// TwinCAT 3 PLC project main
// ProgramVersion: 3.1.4024.0
// libraries:
//   Tc2_Standard, * (Beckhoff Automation GmbH)
//   Tc2_System, * (Beckhoff Automation GmbH)
//   Tc3_Module, * (Beckhoff Automation GmbH)
// project tree:
//   / PlcTask.TcTTO
//   POUs/ MAIN.TcPOU, F_ModbusCrc16.TcPOU, FB_EL6022_Port.TcPOU, FB_ModbusRtuMaster.TcPOU, FB_NimServo.TcPOU, FB_PD33.TcPOU, FB_VibrationSensor.TcPOU
//   GVLs/ GVL_PcDemo.TcGVL, GVL_EL6022_IO.TcGVL, GVL_Rs485Demo.TcGVL, GVL_NimServo.TcGVL, GVL_PD33.TcGVL, GVL_Vibration.TcGVL, GVL_ValveIO.TcGVL, GVL_AnalogSensors.TcGVL, GVL_DataLogger.TcGVL
// real-time tasks:
//   TASK PlcTask: cycle T#2ms, priority 20, ADS port 350
// I/O:
//   DEVICE Device 1 (EtherCAT), AmsNetId 172.24.183.94.2.1
//     Term 7 (EK1200) [EK1200-5000 EtherCAT Power supply (2A E-Bus)]
//       Term 2 (EL1008) [EL1008 8Ch. Dig. Input 24V, 3ms]
//       Term 3 (EL2034) [EL2034 4Ch. Dig. Output 24V, 2A, Diagnostic]
//       Term 4 (EL3742) [EL3742 2Ch. Ana. Input 0-20mA, 16bit, DIFF, Oversample]
//       Term 5 (EL3102) [EL3102 2Ch. Ana. Input +/-10V, Diff.]
//       Term 6 (EL6022) [EL6022 Interface 2Ch. (RS422/485)]
//       Term 13 (EL9011) [EL9011 End Terminal]
//   DEVICE Device 4 (USB)
//     Box 1 (CX2100 Power Supply)
//   DEVICE Device 5 (COM Port)
//   DEVICE Device 6 (NOV-DP-RAM)
// variable links:
//   main/main Instance <-> Device 1 (EtherCAT)/Term 7 (EK1200)/Term 4 (EL3742)
//     PlcTask Inputs/GVL_PcDemo.EL3742_Ch2_Sample0_Raw <-> Ch2 Sample 0/Ch2 Value
//     PlcTask Inputs/GVL_AnalogSensors.Pressure_Raw <-> Ch2 Sample 0/Ch2 Value
//     PlcTask Inputs/GVL_AnalogSensors.Torque_Raw <-> Ch1 Sample 0/Ch1 Value
//   main/main Instance <-> Device 1 (EtherCAT)/Term 7 (EK1200)/Term 3 (EL2034)
//     PlcTask Outputs/GVL_ValveIO.Valve{1..4}_Cmd <-> Channel {1..4}/Output  (4 links)
//   main/main Instance <-> Device 1 (EtherCAT)/Term 7 (EK1200)/Term 6 (EL6022)
//     PlcTask Inputs/GVL_EL6022_IO.EL6022_Ch1_DataIn <-> COM Inputs Channel 1/Data In 0
//     PlcTask Inputs/GVL_EL6022_IO.EL6022_Ch2_DataIn <-> COM Inputs Channel 2/Data In 0
//     PlcTask Inputs/GVL_EL6022_IO.EL6022_Ch1_DataIn @bit 8 <-> COM Inputs Channel 1/Data In 1
//     PlcTask Inputs/GVL_EL6022_IO.EL6022_Ch1_DataIn @bit 80 <-> COM Inputs Channel 1/Data In 10
//     PlcTask Inputs/GVL_EL6022_IO.EL6022_Ch1_DataIn @bit 88 <-> COM Inputs Channel 1/Data In 11
//     PlcTask Inputs/GVL_EL6022_IO.EL6022_Ch1_DataIn @bit 96 <-> COM Inputs Channel 1/Data In 12
//     PlcTask Inputs/GVL_EL6022_IO.EL6022_Ch1_DataIn @bit 104 <-> COM Inputs Channel 1/Data In 13
//     PlcTask Inputs/GVL_EL6022_IO.EL6022_Ch1_DataIn @bit 112 <-> COM Inputs Channel 1/Data In 14
//     PlcTask Inputs/GVL_EL6022_IO.EL6022_Ch1_DataIn @bit 120 <-> COM Inputs Channel 1/Data In 15
//     PlcTask Inputs/GVL_EL6022_IO.EL6022_Ch1_DataIn @bit 128 <-> COM Inputs Channel 1/Data In 16
//     PlcTask Inputs/GVL_EL6022_IO.EL6022_Ch1_DataIn @bit 136 <-> COM Inputs Channel 1/Data In 17
//     PlcTask Inputs/GVL_EL6022_IO.EL6022_Ch1_DataIn @bit 144 <-> COM Inputs Channel 1/Data In 18
//     PlcTask Inputs/GVL_EL6022_IO.EL6022_Ch1_DataIn @bit 152 <-> COM Inputs Channel 1/Data In 19
//     PlcTask Inputs/GVL_EL6022_IO.EL6022_Ch1_DataIn @bit 16 <-> COM Inputs Channel 1/Data In 2
//     PlcTask Inputs/GVL_EL6022_IO.EL6022_Ch1_DataIn @bit 160 <-> COM Inputs Channel 1/Data In 20
//     PlcTask Inputs/GVL_EL6022_IO.EL6022_Ch1_DataIn @bit 168 <-> COM Inputs Channel 1/Data In 21
//     PlcTask Inputs/GVL_EL6022_IO.EL6022_Ch1_DataIn @bit 24 <-> COM Inputs Channel 1/Data In 3
//     PlcTask Inputs/GVL_EL6022_IO.EL6022_Ch1_DataIn @bit 32 <-> COM Inputs Channel 1/Data In 4
//     PlcTask Inputs/GVL_EL6022_IO.EL6022_Ch1_DataIn @bit 40 <-> COM Inputs Channel 1/Data In 5
//     PlcTask Inputs/GVL_EL6022_IO.EL6022_Ch1_DataIn @bit 48 <-> COM Inputs Channel 1/Data In 6
//     PlcTask Inputs/GVL_EL6022_IO.EL6022_Ch1_DataIn @bit 56 <-> COM Inputs Channel 1/Data In 7
//     PlcTask Inputs/GVL_EL6022_IO.EL6022_Ch1_DataIn @bit 64 <-> COM Inputs Channel 1/Data In 8
//     PlcTask Inputs/GVL_EL6022_IO.EL6022_Ch1_DataIn @bit 72 <-> COM Inputs Channel 1/Data In 9
//     PlcTask Inputs/GVL_EL6022_IO.EL6022_Ch2_DataIn @bit 8 <-> COM Inputs Channel 2/Data In 1
//     PlcTask Inputs/GVL_EL6022_IO.EL6022_Ch2_DataIn @bit 80 <-> COM Inputs Channel 2/Data In 10
//     PlcTask Inputs/GVL_EL6022_IO.EL6022_Ch2_DataIn @bit 88 <-> COM Inputs Channel 2/Data In 11
//     PlcTask Inputs/GVL_EL6022_IO.EL6022_Ch2_DataIn @bit 96 <-> COM Inputs Channel 2/Data In 12
//     PlcTask Inputs/GVL_EL6022_IO.EL6022_Ch2_DataIn @bit 104 <-> COM Inputs Channel 2/Data In 13
//     PlcTask Inputs/GVL_EL6022_IO.EL6022_Ch2_DataIn @bit 112 <-> COM Inputs Channel 2/Data In 14
//     PlcTask Inputs/GVL_EL6022_IO.EL6022_Ch2_DataIn @bit 120 <-> COM Inputs Channel 2/Data In 15
//     PlcTask Inputs/GVL_EL6022_IO.EL6022_Ch2_DataIn @bit 128 <-> COM Inputs Channel 2/Data In 16
//     PlcTask Inputs/GVL_EL6022_IO.EL6022_Ch2_DataIn @bit 136 <-> COM Inputs Channel 2/Data In 17
//     PlcTask Inputs/GVL_EL6022_IO.EL6022_Ch2_DataIn @bit 144 <-> COM Inputs Channel 2/Data In 18
//     PlcTask Inputs/GVL_EL6022_IO.EL6022_Ch2_DataIn @bit 152 <-> COM Inputs Channel 2/Data In 19
//     PlcTask Inputs/GVL_EL6022_IO.EL6022_Ch2_DataIn @bit 16 <-> COM Inputs Channel 2/Data In 2
//     PlcTask Inputs/GVL_EL6022_IO.EL6022_Ch2_DataIn @bit 160 <-> COM Inputs Channel 2/Data In 20
//     PlcTask Inputs/GVL_EL6022_IO.EL6022_Ch2_DataIn @bit 168 <-> COM Inputs Channel 2/Data In 21
//     PlcTask Inputs/GVL_EL6022_IO.EL6022_Ch2_DataIn @bit 24 <-> COM Inputs Channel 2/Data In 3
//     PlcTask Inputs/GVL_EL6022_IO.EL6022_Ch2_DataIn @bit 32 <-> COM Inputs Channel 2/Data In 4
//     PlcTask Inputs/GVL_EL6022_IO.EL6022_Ch2_DataIn @bit 40 <-> COM Inputs Channel 2/Data In 5
//     PlcTask Inputs/GVL_EL6022_IO.EL6022_Ch2_DataIn @bit 48 <-> COM Inputs Channel 2/Data In 6
//     PlcTask Inputs/GVL_EL6022_IO.EL6022_Ch2_DataIn @bit 56 <-> COM Inputs Channel 2/Data In 7
//     PlcTask Inputs/GVL_EL6022_IO.EL6022_Ch2_DataIn @bit 64 <-> COM Inputs Channel 2/Data In 8
//     PlcTask Inputs/GVL_EL6022_IO.EL6022_Ch2_DataIn @bit 72 <-> COM Inputs Channel 2/Data In 9
//     PlcTask Inputs/GVL_EL6022_IO.EL6022_Ch1_Status <-> COM Inputs Channel 1/Status
//     PlcTask Inputs/GVL_EL6022_IO.EL6022_Ch2_Status <-> COM Inputs Channel 2/Status
//     PlcTask Outputs/GVL_EL6022_IO.EL6022_Ch1_Ctrl <-> COM Outputs Channel 1/Ctrl
//     PlcTask Outputs/GVL_EL6022_IO.EL6022_Ch2_Ctrl <-> COM Outputs Channel 2/Ctrl
//     PlcTask Outputs/GVL_EL6022_IO.EL6022_Ch1_DataOut <-> COM Outputs Channel 1/Data Out 0
//     PlcTask Outputs/GVL_EL6022_IO.EL6022_Ch2_DataOut <-> COM Outputs Channel 2/Data Out 0
//     PlcTask Outputs/GVL_EL6022_IO.EL6022_Ch1_DataOut @bit 8 <-> COM Outputs Channel 1/Data Out 1
//     PlcTask Outputs/GVL_EL6022_IO.EL6022_Ch1_DataOut @bit 80 <-> COM Outputs Channel 1/Data Out 10
//     PlcTask Outputs/GVL_EL6022_IO.EL6022_Ch1_DataOut @bit 88 <-> COM Outputs Channel 1/Data Out 11
//     PlcTask Outputs/GVL_EL6022_IO.EL6022_Ch1_DataOut @bit 96 <-> COM Outputs Channel 1/Data Out 12
//     PlcTask Outputs/GVL_EL6022_IO.EL6022_Ch1_DataOut @bit 104 <-> COM Outputs Channel 1/Data Out 13
//     PlcTask Outputs/GVL_EL6022_IO.EL6022_Ch1_DataOut @bit 112 <-> COM Outputs Channel 1/Data Out 14
//     PlcTask Outputs/GVL_EL6022_IO.EL6022_Ch1_DataOut @bit 120 <-> COM Outputs Channel 1/Data Out 15
//     PlcTask Outputs/GVL_EL6022_IO.EL6022_Ch1_DataOut @bit 128 <-> COM Outputs Channel 1/Data Out 16
//     PlcTask Outputs/GVL_EL6022_IO.EL6022_Ch1_DataOut @bit 136 <-> COM Outputs Channel 1/Data Out 17
//     PlcTask Outputs/GVL_EL6022_IO.EL6022_Ch1_DataOut @bit 144 <-> COM Outputs Channel 1/Data Out 18
//     PlcTask Outputs/GVL_EL6022_IO.EL6022_Ch1_DataOut @bit 152 <-> COM Outputs Channel 1/Data Out 19
//     PlcTask Outputs/GVL_EL6022_IO.EL6022_Ch1_DataOut @bit 16 <-> COM Outputs Channel 1/Data Out 2
//     PlcTask Outputs/GVL_EL6022_IO.EL6022_Ch1_DataOut @bit 160 <-> COM Outputs Channel 1/Data Out 20
//     PlcTask Outputs/GVL_EL6022_IO.EL6022_Ch1_DataOut @bit 168 <-> COM Outputs Channel 1/Data Out 21
//     PlcTask Outputs/GVL_EL6022_IO.EL6022_Ch1_DataOut @bit 24 <-> COM Outputs Channel 1/Data Out 3
//     PlcTask Outputs/GVL_EL6022_IO.EL6022_Ch1_DataOut @bit 32 <-> COM Outputs Channel 1/Data Out 4
//     PlcTask Outputs/GVL_EL6022_IO.EL6022_Ch1_DataOut @bit 40 <-> COM Outputs Channel 1/Data Out 5
//     PlcTask Outputs/GVL_EL6022_IO.EL6022_Ch1_DataOut @bit 48 <-> COM Outputs Channel 1/Data Out 6
//     PlcTask Outputs/GVL_EL6022_IO.EL6022_Ch1_DataOut @bit 56 <-> COM Outputs Channel 1/Data Out 7
//     PlcTask Outputs/GVL_EL6022_IO.EL6022_Ch1_DataOut @bit 64 <-> COM Outputs Channel 1/Data Out 8
//     PlcTask Outputs/GVL_EL6022_IO.EL6022_Ch1_DataOut @bit 72 <-> COM Outputs Channel 1/Data Out 9
//     PlcTask Outputs/GVL_EL6022_IO.EL6022_Ch2_DataOut @bit 8 <-> COM Outputs Channel 2/Data Out 1
//     PlcTask Outputs/GVL_EL6022_IO.EL6022_Ch2_DataOut @bit 80 <-> COM Outputs Channel 2/Data Out 10
//     PlcTask Outputs/GVL_EL6022_IO.EL6022_Ch2_DataOut @bit 88 <-> COM Outputs Channel 2/Data Out 11
//     PlcTask Outputs/GVL_EL6022_IO.EL6022_Ch2_DataOut @bit 96 <-> COM Outputs Channel 2/Data Out 12
//     PlcTask Outputs/GVL_EL6022_IO.EL6022_Ch2_DataOut @bit 104 <-> COM Outputs Channel 2/Data Out 13
//     PlcTask Outputs/GVL_EL6022_IO.EL6022_Ch2_DataOut @bit 112 <-> COM Outputs Channel 2/Data Out 14
//     PlcTask Outputs/GVL_EL6022_IO.EL6022_Ch2_DataOut @bit 120 <-> COM Outputs Channel 2/Data Out 15
//     PlcTask Outputs/GVL_EL6022_IO.EL6022_Ch2_DataOut @bit 128 <-> COM Outputs Channel 2/Data Out 16
//     PlcTask Outputs/GVL_EL6022_IO.EL6022_Ch2_DataOut @bit 136 <-> COM Outputs Channel 2/Data Out 17
//     PlcTask Outputs/GVL_EL6022_IO.EL6022_Ch2_DataOut @bit 144 <-> COM Outputs Channel 2/Data Out 18
//     PlcTask Outputs/GVL_EL6022_IO.EL6022_Ch2_DataOut @bit 152 <-> COM Outputs Channel 2/Data Out 19
//     PlcTask Outputs/GVL_EL6022_IO.EL6022_Ch2_DataOut @bit 16 <-> COM Outputs Channel 2/Data Out 2
//     PlcTask Outputs/GVL_EL6022_IO.EL6022_Ch2_DataOut @bit 160 <-> COM Outputs Channel 2/Data Out 20
//     PlcTask Outputs/GVL_EL6022_IO.EL6022_Ch2_DataOut @bit 168 <-> COM Outputs Channel 2/Data Out 21
//     PlcTask Outputs/GVL_EL6022_IO.EL6022_Ch2_DataOut @bit 24 <-> COM Outputs Channel 2/Data Out 3
//     PlcTask Outputs/GVL_EL6022_IO.EL6022_Ch2_DataOut @bit 32 <-> COM Outputs Channel 2/Data Out 4
//     PlcTask Outputs/GVL_EL6022_IO.EL6022_Ch2_DataOut @bit 40 <-> COM Outputs Channel 2/Data Out 5
//     PlcTask Outputs/GVL_EL6022_IO.EL6022_Ch2_DataOut @bit 48 <-> COM Outputs Channel 2/Data Out 6
//     PlcTask Outputs/GVL_EL6022_IO.EL6022_Ch2_DataOut @bit 56 <-> COM Outputs Channel 2/Data Out 7
//     PlcTask Outputs/GVL_EL6022_IO.EL6022_Ch2_DataOut @bit 64 <-> COM Outputs Channel 2/Data Out 8
//     PlcTask Outputs/GVL_EL6022_IO.EL6022_Ch2_DataOut @bit 72 <-> COM Outputs Channel 2/Data Out 9

CONFIGURATION main
    RESOURCE PLC ON TwinCAT3
        TASK PlcTask(INTERVAL := T#2ms, PRIORITY := 20);
        PROGRAM MAIN WITH PlcTask : MAIN;
    END_RESOURCE
END_CONFIGURATION

// ---- GVLs/GVL_PcDemo.TcGVL
VAR_GLOBAL
    (*
      Demo input to be linked in TwinCAT I/O mapping:
      EL3742 -> Ch2 Sample 0 -> Ch2 Value
    *)
    EL3742_Ch2_Sample0_Raw AT %I*: INT;

    (*
      PLC-side copy / heartbeat for ADS reads.
    *)
    EL3742_Ch2_Sample0_RawCopy : INT;
    MainCycleCounter : ULINT;
END_VAR

// ---- GVLs/GVL_EL6022_IO.TcGVL
VAR_GLOBAL
    (*
      EL6022 process data mapping placeholders.
      Map these in TwinCAT I/O Mapping to:
        Term 6 (EL6022) -> COM Inputs/Outputs Channel 1/2
      Notes:
        - Status/Ctrl are WORD. Typically: low byte = flags, high byte = length (bytes).
        - Data arrays are 22 bytes (0..21).
    *)

    // Channel 1
    EL6022_Ch1_Status AT %I* : WORD;
    EL6022_Ch1_DataIn AT %I* : ARRAY [0..21] OF USINT;

    EL6022_Ch1_Ctrl AT %Q* : WORD;
    EL6022_Ch1_DataOut AT %Q* : ARRAY [0..21] OF USINT;

    // Channel 2
    EL6022_Ch2_Status AT %I* : WORD;
    EL6022_Ch2_DataIn AT %I* : ARRAY [0..21] OF USINT;

    EL6022_Ch2_Ctrl AT %Q* : WORD;
    EL6022_Ch2_DataOut AT %Q* : ARRAY [0..21] OF USINT;
END_VAR

// ---- GVLs/GVL_Rs485Demo.TcGVL
VAR_GLOBAL
    (*
      PC <-> PLC demo interface for EL6022 RS-485 loopback testing.
      PC writes Tx* and increments TxSeq.
      PLC sends via selected channel and exposes last Rx* from either channel.
    *)

    Enable : BOOL; // Enable demo logic in MAIN (avoid conflicts with real device drivers)

    TxSeq : UDINT;
    TxUseCh2 : BOOL; // FALSE => TX on Ch1, TRUE => TX on Ch2
    TxLen : USINT;
    TxData : ARRAY [0..21] OF USINT;

    TxBusy : BOOL;
    TxDoneSeq : UDINT;
    TxError : UDINT;

    RxSeq : UDINT;
    RxFromCh2 : BOOL;
    RxLen : USINT;
    RxStatus : WORD;
    RxData : ARRAY [0..21] OF USINT;

    Debug_Ch1_Status : WORD;
    Debug_Ch2_Status : WORD;
    Debug_Ch1_Ctrl : WORD;
    Debug_Ch2_Ctrl : WORD;
END_VAR

// ---- GVLs/GVL_NimServo.TcGVL
VAR_GLOBAL
    (*
      NiMotion servo host interface (Modbus RTU over EL6022 / RS-485).

      Notes:
      - PLC implements Modbus + servo control. PC only uses ADS to write macro-level commands and read telemetry.
      - Channel selects EL6022 channel 1/2.
      - WordSwap32 can be used to adapt 32-bit register word order if needed.
    *)

    Enable : BOOL;
    Channel : USINT := 1; // 1 or 2
    SlaveId : USINT := 1; // Modbus address 1..247

    AutoSetCia402Mode : BOOL := TRUE; // Write I2002-1 (H00B1) to 0 if needed

    DesiredMode : USINT := 2; // 2=VM, 9=CSV
    PowerEnable : BOOL;
    TargetVelocity : DINT; // Raw target velocity (unit depends on drive configuration)
    WordSwap32 : BOOL;
    TestForceVelocityWrite : BOOL; // Debug: send 60FF write even without successful comms / OP enabled
    ExtendedPoll : BOOL := TRUE;    // TRUE: poll extended diagnostics (more traffic, more risk of timeouts on noisy links)
    ApplyVmConfig : BOOL := FALSE;  // TRUE: apply VM min/max/accel/decel params via Modbus when PowerEnable=FALSE

    // VM mode parameters (from Modbus.db)
    VmSpeedMinRpm : UDINT := 0;     // I6046-1 (H0385), 32-bit
    VmSpeedMaxRpm : UDINT := 500;   // I6046-2 (H0387), 32-bit
    VmAccelRpm : UDINT := 200;      // I6048-1 (H0389), 32-bit
    VmAccelTimeS : UINT := 1;       // I6048-2 (H038B), 16-bit, seconds
    VmDecelRpm : UDINT := 200;      // I6049-1 (H038C), 32-bit
    VmDecelTimeS : UINT := 1;       // I6049-2 (H038E), 16-bit, seconds

    CmdSeq : UDINT; // PC increments to request a one-shot command
    Cmd : USINT;    // 0=None, 1=FaultReset

    CmdAckSeq : UDINT;
    Busy : BOOL;
    CommOk : BOOL;
    CommErrorCount : UDINT;
    LastErrorId : UDINT;

    // Telemetry (raw registers)
    ControlMode : USINT;      // I2002-1 (H00B1): 0=CIA402
    ControlModeOk : BOOL;
    StatusWord : UINT;         // 6041 (H0381)
    ControlWord : UINT;        // last written 6040 (H0380)

    // Diagnostics / preconditions
    Cia402State : USINT;       // 0=Unknown, 1=NotReady, 2=SwitchOnDisabled, 3=Ready, 4=SwitchedOn, 5=OpEnabled, 6=FaultReaction, 7=Fault, 8=QuickStop
    ErrorRegister : USINT;     // I1001 (H0000) low byte
    CurrentAlarm : USINT;      // I1003-0 (H0001) low byte

    DiSignals : UINT;          // I200B-5 (H01E2), raw DI monitor bits
    DoSignals : UINT;          // I200B-6 (H01E3), raw DO monitor bits
    DcBusVoltage : UINT;       // I200B-21 (H01F7), bus voltage (unit per drive)
    ModuleTemp : INT;          // I200B-22 (H01F8), module temperature (unit per drive)

    Di1Func : USINT;           // I2003-3 (H00D5) low byte
    Di1Logic : USINT;          // I2003-4 (H00D6) low byte
    Di2Func : USINT;           // I2003-5 (H00D7) low byte
    Di2Logic : USINT;          // I2003-6 (H00D8) low byte
    Di3Func : USINT;           // I2003-7 (H00D9) low byte
    Di3Logic : USINT;          // I2003-8 (H00DA) low byte
    Di4Func : USINT;           // I2003-9 (H00DB) low byte
    Di4Logic : USINT;          // I2003-10 (H00DC) low byte
    Di5Func : USINT;           // I2003-11 (H00DD) low byte
    Di5Logic : USINT;          // I2003-12 (H00DE) low byte
    Di6Func : USINT;           // I2003-13 (H00DF) low byte
    Di6Logic : USINT;          // I2003-14 (H00E0) low byte
    Di7Func : USINT;           // I2003-15 (H00E1) low byte
    Di7Logic : USINT;          // I2003-16 (H00E2) low byte
    Di8Func : USINT;           // I2003-17 (H00E3) low byte
    Di8Logic : USINT;          // I2003-18 (H00E4) low byte
    Di9Func : USINT;           // I2003-19 (H00E5) low byte
    Di9Logic : USINT;          // I2003-20 (H00E6) low byte

    EnableDiIndex : USINT;     // 0=None, 1..9 = which DI is "Enable(1)"
    EnableDiRequired : BOOL;   // EnableDiIndex <> 0
    EnableDiActive : BOOL;     // Computed from DiSignals + selected DI logic when required
    EnableDiOk : BOOL;         // NOT EnableDiRequired OR EnableDiActive

    // Drive status (vendor-specific)
    DriveInternalState : USINT; // I200B-1 (H01DE), see Modbus.db selects (0=未准备好, 1=准备好, 8=速度闭环控制...)
    FpgaSystemStatus : UINT;    // I200B-24 (H01FA)
    FpgaSystemFault : UINT;     // I200B-25 (H01FB)
    EncoderInternalFault : UINT; // I200B-26 (H01FC) 编码内部故障信息
    FaultRecord : UINT;         // I200B-27 (H01FD)
    AbsEncoderWord : UINT;      // I200B-23 (H01F9) FPGA给出绝对编码

    ModeDisplay : USINT;       // 6061 (H03C3) low byte
    ActualVelocity : DINT;     // 606C (H03D5)
    ActualPosition : DINT;     // 6064 (H03C8)
    CurrentFeedback : INT;     // 6078 (H03E4)

    // VM mode telemetry (from Modbus.db)
    VmTargetSpeedRpm : INT;    // I6042 (H0382) 16-bit
    VmTargetSpeedEffRpm : INT; // I6043 (H0383) 16-bit (effective)
    VmActualSpeedRpm : INT;    // I6044 (H0384) 16-bit

    // VM config progress (helps debug/avoid powering on before config is applied)
    VmCfgPending : BOOL;
    VmCfgIndex : USINT;

    // Debug frames
    LastTxLen : USINT;
    LastTx : ARRAY [0..21] OF USINT;
    LastRxLen : USINT;
    LastRx : ARRAY [0..21] OF USINT;
END_VAR

// ---- GVLs/GVL_PD33.TcGVL
VAR_GLOBAL
    (*
      PD33 series laser displacement sensor (Modbus RTU over EL6022 / RS-485).

      Registers (from manual screenshots):
      Current mode: passive parsing of PD33 full-speed active output.
      Expected frame: slave=1, function=3, bytecount=4, payload i32 low-word-first, CRC16.
      Scale: raw / 1000.0 = mm.
    *)

    Enable : BOOL;
    Channel : USINT := 1; // 1 or 2 (EL6022 channel)
    SlaveId : USINT := 1; // Modbus address

    // PD33 frames shown in the manual interpret 32-bit values as "low word first".
    // Keep this TRUE unless you verify your device uses the opposite order.
    WordSwap32 : BOOL := TRUE;
    UseDisplayRegister3B : BOOL := FALSE; // reserved; passive full-speed output parser does not send read requests

    // Command handshake (PC writes Cmd+CmdSeq; PLC sets CmdAckSeq after completion)
    CmdSeq : UDINT;
    Cmd : USINT; // reserved in passive mode
    CmdAckSeq : UDINT;
    Busy : BOOL;

    // Diagnostics
    ChannelConflict : BOOL; // TRUE when another driver is using the same EL6022 channel
    PortReady : BOOL;
    CommOk : BOOL;
    CommErrorCount : UDINT;
    LastErrorId : UDINT;
    ExceptionCode : USINT;
    RxDiscardCount : UDINT;
    LastDiscardId : UDINT;

    // Measurements
    AbsRaw : DINT; // raw units depend on UseDisplayRegister3B
    RelRaw : DINT; // raw units depend on UseDisplayRegister3B
    AbsMm : LREAL; // computed
    RelMm : LREAL; // computed

    ZeroWord : UINT; // last written value to 0x0020 (for debug)

    // Debug frames (last Modbus tx/rx)
    LastTxLen : USINT;
    LastTx : ARRAY [0..21] OF USINT;
    LastRxLen : USINT;
    LastRx : ARRAY [0..21] OF USINT;
END_VAR

// ---- GVLs/GVL_Vibration.TcGVL
VAR_GLOBAL
    (*
      VB02/WTVB02-485 vibration sensor over EL6022 Channel 2.

      SDK register map:
        0x34..0x36 vibration acceleration X/Y/Z, raw INT, scale raw / 32768 * 16
        0x3A..0x3C vibration velocity X/Y/Z, raw INT, scale raw / 100
        0x40      temperature, raw INT, scale raw / 100
        0x41..0x43 displacement X/Y/Z, raw INT
        0x44..0x46 frequency X/Y/Z, raw INT, scale raw / 10

      EL6022 frame limit is 22 bytes, so PLC reads these as 3 Modbus transactions.
    *)

    Enable : BOOL := FALSE;
    Channel : USINT := 2;
    SlaveId : USINT := 16#50;
    MinGapMs : UINT := 200;
    TimeoutMs : UINT := 500;

    Busy : BOOL;
    PortReady : BOOL;
    CommOk : BOOL;
    CommErrorCount : UDINT;
    LastErrorId : UDINT;
    ExceptionCode : USINT;
    RxDiscardCount : UDINT;
    LastDiscardId : UDINT;
    SampleSeq : UDINT;

    AccXRaw : INT;
    AccYRaw : INT;
    AccZRaw : INT;
    VelXRaw : INT;
    VelYRaw : INT;
    VelZRaw : INT;
    TempRaw : INT;
    DispXRaw : INT;
    DispYRaw : INT;
    DispZRaw : INT;
    FreqXRaw : INT;
    FreqYRaw : INT;
    FreqZRaw : INT;

    AccX : LREAL;
    AccY : LREAL;
    AccZ : LREAL;
    VelX : LREAL;
    VelY : LREAL;
    VelZ : LREAL;
    TempC : LREAL;
    DispX : LREAL;
    DispY : LREAL;
    DispZ : LREAL;
    FreqX : LREAL;
    FreqY : LREAL;
    FreqZ : LREAL;

    LastTxLen : USINT;
    LastTx : ARRAY [0..21] OF USINT;
    LastRxLen : USINT;
    LastRx : ARRAY [0..21] OF USINT;
END_VAR

// ---- GVLs/GVL_ValveIO.TcGVL
VAR_GLOBAL
    (*
      Valve digital outputs placeholder.

      Hardware: Term 3 (EL2034) 4Ch. Digital Output.

      Map in TwinCAT I/O mapping:
        EL2034 -> Channel 1 -> Output  => Valve1_Cmd
        EL2034 -> Channel 2 -> Output  => Valve2_Cmd
        EL2034 -> Channel 3 -> Output  => Valve3_Cmd
        EL2034 -> Channel 4 -> Output  => Valve4_Cmd

      Notes:
        - Use AT %Q* so the symbol shows up in "Link To..." list.
        - Valve*_Fb are software feedback mirrors (what PLC currently drives).
    *)

    Valve1_Cmd AT %Q* : BOOL;
    Valve2_Cmd AT %Q* : BOOL;
    Valve3_Cmd AT %Q* : BOOL;
    Valve4_Cmd AT %Q* : BOOL;

    Valve1_Fb : BOOL;
    Valve2_Fb : BOOL;
    Valve3_Fb : BOOL;
    Valve4_Fb : BOOL;

    // Master enable for all valve outputs (safety interlock).
    Enable : BOOL := FALSE;
END_VAR

// ---- GVLs/GVL_AnalogSensors.TcGVL
VAR_GLOBAL
    (*
      Analog current sampling (EL3742 2Ch 0-20mA) placeholders.

      Map in TwinCAT I/O mapping:
        EL3742 -> Ch2 Sample 0 -> Ch2 Value => Pressure_Raw
        EL3742 -> Ch1 Sample 0 -> Ch1 Value => Torque_Raw

      Raw type follows EL3742 PDO type (INT16).
    *)

    Pressure_Raw AT %I* : INT;
    Torque_Raw AT %I* : INT;

    // PLC-side copies for ADS reads / snapshot.
    Pressure_RawCopy : INT;
    Torque_RawCopy : INT;
END_VAR

// ---- GVLs/GVL_DataLogger.TcGVL
VAR_GLOBAL
    (*
      PLC-side ring buffer logger to avoid ADS per-sample reads.

      Design:
        - MAIN (2ms task) writes a fixed-size record into a byte ring buffer.
        - PC reads Head and Buffer bytes via ADS and reconstructs records.
        - If PC is too slow and overrun happens, OverrunCount increments.

      Record layout (little-endian):
        u32 magic = 0x56424D31 ('VBM1')
        u32 seq
        u32 t_us (monotonic from cycle count * 2000us)
        i16 pressure_raw
        i16 torque_raw
        i32 pd33_abs_raw
        i32 pd33_rel_raw
        i16 vib_acc_x_raw
        i16 vib_acc_y_raw
        i16 vib_acc_z_raw
        i16 vib_vel_x_raw
        i16 vib_vel_y_raw
        i16 vib_vel_z_raw
        i16 vib_temp_raw
        i16 vib_disp_x_raw
        i16 vib_disp_y_raw
        i16 vib_disp_z_raw
        i16 vib_freq_x_raw
        i16 vib_freq_y_raw
        i16 vib_freq_z_raw
        u8  valves (bit0..3)
        u8  flags (bit0=pd33_comm_ok, bit1=vibration_comm_ok)
        u16 reserved
      Total: 54 bytes per record
    *)

    Enable : BOOL := FALSE;
    Reset : BOOL := FALSE;

    // Ring buffer state (byte indices)
    Head : UDINT; // next write index (monotonic, wraps by modulo on read side)
    Tail : UDINT; // PC should update this as "consumed" index to prevent Overrun

    OverrunCount : UDINT;
    DropCount : UDINT;

    Seq : UDINT;

    // Constants
    RecordSize : UDINT := 54;
    BufferSize : UDINT := 54 * 4096; // 221,184 bytes (~8.2s at 500Hz)

    Buffer : ARRAY [0..(54*4096)-1] OF USINT;
END_VAR

// ---- POUs/MAIN.TcPOU
PROGRAM MAIN
VAR
    initCh1Done : BOOL;
    initCh2Done : BOOL;
    fbNimServo : FB_NimServo;
    fbPd33 : FB_PD33;
    fbVibration : FB_VibrationSensor;

    // DataLogger internal (packed ring buffer)
    logResetLatched : BOOL;
    rec : ARRAY [0..53] OF USINT;
    base : UDINT;
    headMod : UDINT;
    seqLocal : UDINT;
    tUs : UDINT;
    tmpU32 : UDINT;
    tmpI16 : INT;
    tmpI32 : DINT;
    valvesBits : USINT;
END_VAR

GVL_PcDemo.MainCycleCounter := GVL_PcDemo.MainCycleCounter + 1;
GVL_PcDemo.EL3742_Ch2_Sample0_RawCopy := GVL_PcDemo.EL3742_Ch2_Sample0_Raw;

// --- Valve digital outputs (EL2034) ---
IF NOT GVL_ValveIO.Enable THEN
    GVL_ValveIO.Valve1_Cmd := FALSE;
    GVL_ValveIO.Valve2_Cmd := FALSE;
    GVL_ValveIO.Valve3_Cmd := FALSE;
    GVL_ValveIO.Valve4_Cmd := FALSE;
END_IF
GVL_ValveIO.Valve1_Fb := GVL_ValveIO.Valve1_Cmd;
GVL_ValveIO.Valve2_Fb := GVL_ValveIO.Valve2_Cmd;
GVL_ValveIO.Valve3_Fb := GVL_ValveIO.Valve3_Cmd;
GVL_ValveIO.Valve4_Fb := GVL_ValveIO.Valve4_Cmd;

// --- Analog sensors (EL3742) ---
GVL_AnalogSensors.Pressure_RawCopy := GVL_AnalogSensors.Pressure_Raw;
GVL_AnalogSensors.Torque_RawCopy := GVL_AnalogSensors.Torque_Raw;

// Keep EL6022 debug always updated (used by PcHostConsole el6022-dump)
GVL_Rs485Demo.Debug_Ch1_Status := GVL_EL6022_IO.EL6022_Ch1_Status;
GVL_Rs485Demo.Debug_Ch2_Status := GVL_EL6022_IO.EL6022_Ch2_Status;
GVL_Rs485Demo.Debug_Ch1_Ctrl := GVL_EL6022_IO.EL6022_Ch1_Ctrl;
GVL_Rs485Demo.Debug_Ch2_Ctrl := GVL_EL6022_IO.EL6022_Ch2_Ctrl;

// --- NiMotion servo (Modbus RTU over EL6022 / RS-485) ---
fbNimServo(
    Enable := GVL_NimServo.Enable,
    Channel := GVL_NimServo.Channel,
    SlaveId := GVL_NimServo.SlaveId,
    AutoSetCia402Mode := GVL_NimServo.AutoSetCia402Mode,
    DesiredMode := GVL_NimServo.DesiredMode,
    PowerEnable := GVL_NimServo.PowerEnable,
    TargetVelocity := GVL_NimServo.TargetVelocity,
    WordSwap32 := GVL_NimServo.WordSwap32,
    TestForceVelocityWrite := GVL_NimServo.TestForceVelocityWrite,
    ExtendedPoll := GVL_NimServo.ExtendedPoll,
    ApplyVmConfig := GVL_NimServo.ApplyVmConfig,
    VmSpeedMinRpm := GVL_NimServo.VmSpeedMinRpm,
    VmSpeedMaxRpm := GVL_NimServo.VmSpeedMaxRpm,
    VmAccelRpm := GVL_NimServo.VmAccelRpm,
    VmAccelTimeS := GVL_NimServo.VmAccelTimeS,
    VmDecelRpm := GVL_NimServo.VmDecelRpm,
    VmDecelTimeS := GVL_NimServo.VmDecelTimeS,
    CmdSeq := GVL_NimServo.CmdSeq,
    Cmd := GVL_NimServo.Cmd
);

GVL_NimServo.CmdAckSeq := fbNimServo.CmdAckSeq;
GVL_NimServo.Busy := fbNimServo.Busy;
GVL_NimServo.CommOk := fbNimServo.CommOk;
GVL_NimServo.CommErrorCount := fbNimServo.CommErrorCount;
GVL_NimServo.LastErrorId := fbNimServo.LastErrorId;
GVL_NimServo.ControlMode := fbNimServo.ControlMode;
GVL_NimServo.ControlModeOk := fbNimServo.ControlModeOk;
GVL_NimServo.StatusWord := fbNimServo.StatusWord;
GVL_NimServo.ControlWord := fbNimServo.ControlWord;
GVL_NimServo.Cia402State := fbNimServo.Cia402State;
GVL_NimServo.ErrorRegister := fbNimServo.ErrorRegister;
GVL_NimServo.CurrentAlarm := fbNimServo.CurrentAlarm;
GVL_NimServo.DiSignals := fbNimServo.DiSignals;
GVL_NimServo.DoSignals := fbNimServo.DoSignals;
GVL_NimServo.DcBusVoltage := fbNimServo.DcBusVoltage;
GVL_NimServo.ModuleTemp := fbNimServo.ModuleTemp;
GVL_NimServo.Di1Func := fbNimServo.Di1Func;
GVL_NimServo.Di1Logic := fbNimServo.Di1Logic;
GVL_NimServo.Di2Func := fbNimServo.Di2Func;
GVL_NimServo.Di2Logic := fbNimServo.Di2Logic;
GVL_NimServo.Di3Func := fbNimServo.Di3Func;
GVL_NimServo.Di3Logic := fbNimServo.Di3Logic;
GVL_NimServo.Di4Func := fbNimServo.Di4Func;
GVL_NimServo.Di4Logic := fbNimServo.Di4Logic;
GVL_NimServo.Di5Func := fbNimServo.Di5Func;
GVL_NimServo.Di5Logic := fbNimServo.Di5Logic;
GVL_NimServo.Di6Func := fbNimServo.Di6Func;
GVL_NimServo.Di6Logic := fbNimServo.Di6Logic;
GVL_NimServo.Di7Func := fbNimServo.Di7Func;
GVL_NimServo.Di7Logic := fbNimServo.Di7Logic;
GVL_NimServo.Di8Func := fbNimServo.Di8Func;
GVL_NimServo.Di8Logic := fbNimServo.Di8Logic;
GVL_NimServo.Di9Func := fbNimServo.Di9Func;
GVL_NimServo.Di9Logic := fbNimServo.Di9Logic;
GVL_NimServo.EnableDiIndex := fbNimServo.EnableDiIndex;
GVL_NimServo.EnableDiRequired := fbNimServo.EnableDiRequired;
GVL_NimServo.EnableDiActive := fbNimServo.EnableDiActive;
GVL_NimServo.EnableDiOk := fbNimServo.EnableDiOk;
GVL_NimServo.DriveInternalState := fbNimServo.DriveInternalState;
GVL_NimServo.FpgaSystemStatus := fbNimServo.FpgaSystemStatus;
GVL_NimServo.FpgaSystemFault := fbNimServo.FpgaSystemFault;
GVL_NimServo.EncoderInternalFault := fbNimServo.EncoderInternalFault;
GVL_NimServo.FaultRecord := fbNimServo.FaultRecord;
GVL_NimServo.AbsEncoderWord := fbNimServo.AbsEncoderWord;
GVL_NimServo.ModeDisplay := fbNimServo.ModeDisplay;
GVL_NimServo.ActualVelocity := fbNimServo.ActualVelocity;
GVL_NimServo.ActualPosition := fbNimServo.ActualPosition;
GVL_NimServo.CurrentFeedback := fbNimServo.CurrentFeedback;
GVL_NimServo.VmTargetSpeedRpm := fbNimServo.VmTargetSpeedRpm;
GVL_NimServo.VmTargetSpeedEffRpm := fbNimServo.VmTargetSpeedEffRpm;
GVL_NimServo.VmActualSpeedRpm := fbNimServo.VmActualSpeedRpm;
GVL_NimServo.VmCfgPending := fbNimServo.VmCfgPendingOut;
GVL_NimServo.VmCfgIndex := fbNimServo.VmCfgIndexOut;
GVL_NimServo.LastTxLen := fbNimServo.LastTxLen;
GVL_NimServo.LastTx := fbNimServo.LastTx;
GVL_NimServo.LastRxLen := fbNimServo.LastRxLen;
GVL_NimServo.LastRx := fbNimServo.LastRx;

// --- PD33 laser displacement sensor (Modbus RTU over EL6022 / RS-485) ---
GVL_PD33.ChannelConflict := GVL_PD33.Enable AND GVL_NimServo.Enable AND (GVL_PD33.Channel = GVL_NimServo.Channel);
fbPd33(
    Enable := GVL_PD33.Enable AND (NOT GVL_PD33.ChannelConflict),
    Channel := GVL_PD33.Channel,
    SlaveId := GVL_PD33.SlaveId,
    WordSwap32 := GVL_PD33.WordSwap32,
    UseDisplayRegister3B := GVL_PD33.UseDisplayRegister3B,
    CmdSeq := GVL_PD33.CmdSeq,
    Cmd := GVL_PD33.Cmd
);
GVL_PD33.CmdAckSeq := fbPd33.CmdAckSeq;
GVL_PD33.Busy := fbPd33.Busy;
GVL_PD33.PortReady := fbPd33.PortReady;
GVL_PD33.CommOk := fbPd33.CommOk;
GVL_PD33.CommErrorCount := fbPd33.CommErrorCount;
GVL_PD33.LastErrorId := fbPd33.LastErrorId;
GVL_PD33.ExceptionCode := fbPd33.ExceptionCode;
GVL_PD33.RxDiscardCount := fbPd33.RxDiscardCount;
GVL_PD33.LastDiscardId := fbPd33.LastDiscardId;
GVL_PD33.AbsRaw := fbPd33.AbsRaw;
GVL_PD33.RelRaw := fbPd33.RelRaw;
GVL_PD33.AbsMm := fbPd33.AbsMm;
GVL_PD33.RelMm := fbPd33.RelMm;
GVL_PD33.ZeroWord := fbPd33.ZeroWord;
GVL_PD33.LastTxLen := fbPd33.LastTxLen;
GVL_PD33.LastTx := fbPd33.LastTx;
GVL_PD33.LastRxLen := fbPd33.LastRxLen;
GVL_PD33.LastRx := fbPd33.LastRx;

// --- VB02 vibration sensor (Modbus RTU over EL6022 Ch2 / RS-485) ---
fbVibration(
    Enable := GVL_Vibration.Enable,
    Channel := GVL_Vibration.Channel,
    SlaveId := GVL_Vibration.SlaveId,
    MinGapMs := GVL_Vibration.MinGapMs,
    TimeoutMs := GVL_Vibration.TimeoutMs
);
GVL_Vibration.Busy := fbVibration.Busy;
GVL_Vibration.PortReady := fbVibration.PortReady;
GVL_Vibration.CommOk := fbVibration.CommOk;
GVL_Vibration.CommErrorCount := fbVibration.CommErrorCount;
GVL_Vibration.LastErrorId := fbVibration.LastErrorId;
GVL_Vibration.ExceptionCode := fbVibration.ExceptionCode;
GVL_Vibration.RxDiscardCount := fbVibration.RxDiscardCount;
GVL_Vibration.LastDiscardId := fbVibration.LastDiscardId;
GVL_Vibration.SampleSeq := fbVibration.SampleSeq;
GVL_Vibration.AccXRaw := fbVibration.AccXRaw;
GVL_Vibration.AccYRaw := fbVibration.AccYRaw;
GVL_Vibration.AccZRaw := fbVibration.AccZRaw;
GVL_Vibration.VelXRaw := fbVibration.VelXRaw;
GVL_Vibration.VelYRaw := fbVibration.VelYRaw;
GVL_Vibration.VelZRaw := fbVibration.VelZRaw;
GVL_Vibration.TempRaw := fbVibration.TempRaw;
GVL_Vibration.DispXRaw := fbVibration.DispXRaw;
GVL_Vibration.DispYRaw := fbVibration.DispYRaw;
GVL_Vibration.DispZRaw := fbVibration.DispZRaw;
GVL_Vibration.FreqXRaw := fbVibration.FreqXRaw;
GVL_Vibration.FreqYRaw := fbVibration.FreqYRaw;
GVL_Vibration.FreqZRaw := fbVibration.FreqZRaw;
GVL_Vibration.AccX := fbVibration.AccX;
GVL_Vibration.AccY := fbVibration.AccY;
GVL_Vibration.AccZ := fbVibration.AccZ;
GVL_Vibration.VelX := fbVibration.VelX;
GVL_Vibration.VelY := fbVibration.VelY;
GVL_Vibration.VelZ := fbVibration.VelZ;
GVL_Vibration.TempC := fbVibration.TempC;
GVL_Vibration.DispX := fbVibration.DispX;
GVL_Vibration.DispY := fbVibration.DispY;
GVL_Vibration.DispZ := fbVibration.DispZ;
GVL_Vibration.FreqX := fbVibration.FreqX;
GVL_Vibration.FreqY := fbVibration.FreqY;
GVL_Vibration.FreqZ := fbVibration.FreqZ;
GVL_Vibration.LastTxLen := fbVibration.LastTxLen;
GVL_Vibration.LastTx := fbVibration.LastTx;
GVL_Vibration.LastRxLen := fbVibration.LastRxLen;
GVL_Vibration.LastRx := fbVibration.LastRx;
// --- DataLogger ring buffer (packed bytes) ---
// Time base: PlcTask cycle is 2000us (see PlcTask.TcTTO). Use cycle counter for monotonic time.
tUs := ULINT_TO_UDINT(GVL_PcDemo.MainCycleCounter) * 2000;

IF GVL_DataLogger.Reset AND (NOT logResetLatched) THEN
    logResetLatched := TRUE;
    GVL_DataLogger.Head := 0;
    GVL_DataLogger.Tail := 0;
    GVL_DataLogger.Seq := 0;
    GVL_DataLogger.OverrunCount := 0;
    GVL_DataLogger.DropCount := 0;
ELSIF (NOT GVL_DataLogger.Reset) THEN
    logResetLatched := FALSE;
END_IF

IF GVL_DataLogger.Enable THEN
    // Overrun detection: if head - tail > BufferSize - RecordSize, drop this sample.
    IF (GVL_DataLogger.Head - GVL_DataLogger.Tail) > (GVL_DataLogger.BufferSize - GVL_DataLogger.RecordSize) THEN
        GVL_DataLogger.OverrunCount := GVL_DataLogger.OverrunCount + 1;
    ELSE
        seqLocal := GVL_DataLogger.Seq;

        // magic 'VBM1' = 0x56424D31
        rec[0] := 16#31; rec[1] := 16#4D; rec[2] := 16#42; rec[3] := 16#56;

        // seq (u32)
        tmpU32 := seqLocal;
        rec[4] := UDINT_TO_USINT(tmpU32 AND 16#FF);
        rec[5] := UDINT_TO_USINT(SHR(tmpU32, 8) AND 16#FF);
        rec[6] := UDINT_TO_USINT(SHR(tmpU32, 16) AND 16#FF);
        rec[7] := UDINT_TO_USINT(SHR(tmpU32, 24) AND 16#FF);

        // t_us (u32)
        tmpU32 := tUs;
        rec[8] := UDINT_TO_USINT(tmpU32 AND 16#FF);
        rec[9] := UDINT_TO_USINT(SHR(tmpU32, 8) AND 16#FF);
        rec[10] := UDINT_TO_USINT(SHR(tmpU32, 16) AND 16#FF);
        rec[11] := UDINT_TO_USINT(SHR(tmpU32, 24) AND 16#FF);

        // pressure_raw (i16)
        tmpI16 := GVL_AnalogSensors.Pressure_RawCopy;
        tmpU32 := INT_TO_UDINT(tmpI16) AND 16#FFFF;
        rec[12] := UDINT_TO_USINT(tmpU32 AND 16#FF);
        rec[13] := UDINT_TO_USINT(SHR(tmpU32, 8) AND 16#FF);

        // torque_raw (i16)
        tmpI16 := GVL_AnalogSensors.Torque_RawCopy;
        tmpU32 := INT_TO_UDINT(tmpI16) AND 16#FFFF;
        rec[14] := UDINT_TO_USINT(tmpU32 AND 16#FF);
        rec[15] := UDINT_TO_USINT(SHR(tmpU32, 8) AND 16#FF);

        // pd33_abs_raw (i32)
        tmpI32 := GVL_PD33.AbsRaw;
        tmpU32 := DINT_TO_UDINT(tmpI32);
        rec[16] := UDINT_TO_USINT(tmpU32 AND 16#FF);
        rec[17] := UDINT_TO_USINT(SHR(tmpU32, 8) AND 16#FF);
        rec[18] := UDINT_TO_USINT(SHR(tmpU32, 16) AND 16#FF);
        rec[19] := UDINT_TO_USINT(SHR(tmpU32, 24) AND 16#FF);

        // pd33_rel_raw (i32)
        tmpI32 := GVL_PD33.RelRaw;
        tmpU32 := DINT_TO_UDINT(tmpI32);
        rec[20] := UDINT_TO_USINT(tmpU32 AND 16#FF);
        rec[21] := UDINT_TO_USINT(SHR(tmpU32, 8) AND 16#FF);
        rec[22] := UDINT_TO_USINT(SHR(tmpU32, 16) AND 16#FF);
        rec[23] := UDINT_TO_USINT(SHR(tmpU32, 24) AND 16#FF);

        // vibration raw values (i16)
        tmpI16 := GVL_Vibration.AccXRaw;
        tmpU32 := INT_TO_UDINT(tmpI16) AND 16#FFFF;
        rec[24] := UDINT_TO_USINT(tmpU32 AND 16#FF);
        rec[25] := UDINT_TO_USINT(SHR(tmpU32, 8) AND 16#FF);

        tmpI16 := GVL_Vibration.AccYRaw;
        tmpU32 := INT_TO_UDINT(tmpI16) AND 16#FFFF;
        rec[26] := UDINT_TO_USINT(tmpU32 AND 16#FF);
        rec[27] := UDINT_TO_USINT(SHR(tmpU32, 8) AND 16#FF);

        tmpI16 := GVL_Vibration.AccZRaw;
        tmpU32 := INT_TO_UDINT(tmpI16) AND 16#FFFF;
        rec[28] := UDINT_TO_USINT(tmpU32 AND 16#FF);
        rec[29] := UDINT_TO_USINT(SHR(tmpU32, 8) AND 16#FF);

        tmpI16 := GVL_Vibration.VelXRaw;
        tmpU32 := INT_TO_UDINT(tmpI16) AND 16#FFFF;
        rec[30] := UDINT_TO_USINT(tmpU32 AND 16#FF);
        rec[31] := UDINT_TO_USINT(SHR(tmpU32, 8) AND 16#FF);

        tmpI16 := GVL_Vibration.VelYRaw;
        tmpU32 := INT_TO_UDINT(tmpI16) AND 16#FFFF;
        rec[32] := UDINT_TO_USINT(tmpU32 AND 16#FF);
        rec[33] := UDINT_TO_USINT(SHR(tmpU32, 8) AND 16#FF);

        tmpI16 := GVL_Vibration.VelZRaw;
        tmpU32 := INT_TO_UDINT(tmpI16) AND 16#FFFF;
        rec[34] := UDINT_TO_USINT(tmpU32 AND 16#FF);
        rec[35] := UDINT_TO_USINT(SHR(tmpU32, 8) AND 16#FF);

        tmpI16 := GVL_Vibration.TempRaw;
        tmpU32 := INT_TO_UDINT(tmpI16) AND 16#FFFF;
        rec[36] := UDINT_TO_USINT(tmpU32 AND 16#FF);
        rec[37] := UDINT_TO_USINT(SHR(tmpU32, 8) AND 16#FF);

        tmpI16 := GVL_Vibration.DispXRaw;
        tmpU32 := INT_TO_UDINT(tmpI16) AND 16#FFFF;
        rec[38] := UDINT_TO_USINT(tmpU32 AND 16#FF);
        rec[39] := UDINT_TO_USINT(SHR(tmpU32, 8) AND 16#FF);

        tmpI16 := GVL_Vibration.DispYRaw;
        tmpU32 := INT_TO_UDINT(tmpI16) AND 16#FFFF;
        rec[40] := UDINT_TO_USINT(tmpU32 AND 16#FF);
        rec[41] := UDINT_TO_USINT(SHR(tmpU32, 8) AND 16#FF);

        tmpI16 := GVL_Vibration.DispZRaw;
        tmpU32 := INT_TO_UDINT(tmpI16) AND 16#FFFF;
        rec[42] := UDINT_TO_USINT(tmpU32 AND 16#FF);
        rec[43] := UDINT_TO_USINT(SHR(tmpU32, 8) AND 16#FF);

        tmpI16 := GVL_Vibration.FreqXRaw;
        tmpU32 := INT_TO_UDINT(tmpI16) AND 16#FFFF;
        rec[44] := UDINT_TO_USINT(tmpU32 AND 16#FF);
        rec[45] := UDINT_TO_USINT(SHR(tmpU32, 8) AND 16#FF);

        tmpI16 := GVL_Vibration.FreqYRaw;
        tmpU32 := INT_TO_UDINT(tmpI16) AND 16#FFFF;
        rec[46] := UDINT_TO_USINT(tmpU32 AND 16#FF);
        rec[47] := UDINT_TO_USINT(SHR(tmpU32, 8) AND 16#FF);

        tmpI16 := GVL_Vibration.FreqZRaw;
        tmpU32 := INT_TO_UDINT(tmpI16) AND 16#FFFF;
        rec[48] := UDINT_TO_USINT(tmpU32 AND 16#FF);
        rec[49] := UDINT_TO_USINT(SHR(tmpU32, 8) AND 16#FF);
        // valves bits
        valvesBits := 0;
        IF GVL_ValveIO.Valve1_Fb THEN valvesBits := valvesBits OR 16#01; END_IF
        IF GVL_ValveIO.Valve2_Fb THEN valvesBits := valvesBits OR 16#02; END_IF
        IF GVL_ValveIO.Valve3_Fb THEN valvesBits := valvesBits OR 16#04; END_IF
        IF GVL_ValveIO.Valve4_Fb THEN valvesBits := valvesBits OR 16#08; END_IF
        rec[50] := valvesBits;

        // flags
        rec[51] := 0;
        IF GVL_PD33.CommOk THEN rec[51] := rec[51] OR 16#01; END_IF
        IF GVL_Vibration.CommOk THEN rec[51] := rec[51] OR 16#02; END_IF

        // reserved u16
        rec[52] := 0;
        rec[53] := 0;

        // write record into ring (buffer size is multiple of record size)
        headMod := GVL_DataLogger.Head MOD GVL_DataLogger.BufferSize;
        base := headMod;
        GVL_DataLogger.Buffer[base + 0] := rec[0];
        GVL_DataLogger.Buffer[base + 1] := rec[1];
        GVL_DataLogger.Buffer[base + 2] := rec[2];
        GVL_DataLogger.Buffer[base + 3] := rec[3];
        GVL_DataLogger.Buffer[base + 4] := rec[4];
        GVL_DataLogger.Buffer[base + 5] := rec[5];
        GVL_DataLogger.Buffer[base + 6] := rec[6];
        GVL_DataLogger.Buffer[base + 7] := rec[7];
        GVL_DataLogger.Buffer[base + 8] := rec[8];
        GVL_DataLogger.Buffer[base + 9] := rec[9];
        GVL_DataLogger.Buffer[base + 10] := rec[10];
        GVL_DataLogger.Buffer[base + 11] := rec[11];
        GVL_DataLogger.Buffer[base + 12] := rec[12];
        GVL_DataLogger.Buffer[base + 13] := rec[13];
        GVL_DataLogger.Buffer[base + 14] := rec[14];
        GVL_DataLogger.Buffer[base + 15] := rec[15];
        GVL_DataLogger.Buffer[base + 16] := rec[16];
        GVL_DataLogger.Buffer[base + 17] := rec[17];
        GVL_DataLogger.Buffer[base + 18] := rec[18];
        GVL_DataLogger.Buffer[base + 19] := rec[19];
        GVL_DataLogger.Buffer[base + 20] := rec[20];
        GVL_DataLogger.Buffer[base + 21] := rec[21];
        GVL_DataLogger.Buffer[base + 22] := rec[22];
        GVL_DataLogger.Buffer[base + 23] := rec[23];
        GVL_DataLogger.Buffer[base + 24] := rec[24];
        GVL_DataLogger.Buffer[base + 25] := rec[25];
        GVL_DataLogger.Buffer[base + 26] := rec[26];
        GVL_DataLogger.Buffer[base + 27] := rec[27];
        GVL_DataLogger.Buffer[base + 28] := rec[28];
        GVL_DataLogger.Buffer[base + 29] := rec[29];
        GVL_DataLogger.Buffer[base + 30] := rec[30];
        GVL_DataLogger.Buffer[base + 31] := rec[31];
        GVL_DataLogger.Buffer[base + 32] := rec[32];
        GVL_DataLogger.Buffer[base + 33] := rec[33];
        GVL_DataLogger.Buffer[base + 34] := rec[34];
        GVL_DataLogger.Buffer[base + 35] := rec[35];
        GVL_DataLogger.Buffer[base + 36] := rec[36];
        GVL_DataLogger.Buffer[base + 37] := rec[37];
        GVL_DataLogger.Buffer[base + 38] := rec[38];
        GVL_DataLogger.Buffer[base + 39] := rec[39];
        GVL_DataLogger.Buffer[base + 40] := rec[40];
        GVL_DataLogger.Buffer[base + 41] := rec[41];
        GVL_DataLogger.Buffer[base + 42] := rec[42];
        GVL_DataLogger.Buffer[base + 43] := rec[43];
        GVL_DataLogger.Buffer[base + 44] := rec[44];
        GVL_DataLogger.Buffer[base + 45] := rec[45];
        GVL_DataLogger.Buffer[base + 46] := rec[46];
        GVL_DataLogger.Buffer[base + 47] := rec[47];
        GVL_DataLogger.Buffer[base + 48] := rec[48];
        GVL_DataLogger.Buffer[base + 49] := rec[49];
        GVL_DataLogger.Buffer[base + 50] := rec[50];
        GVL_DataLogger.Buffer[base + 51] := rec[51];
        GVL_DataLogger.Buffer[base + 52] := rec[52];
        GVL_DataLogger.Buffer[base + 53] := rec[53];

        GVL_DataLogger.Head := GVL_DataLogger.Head + GVL_DataLogger.RecordSize;
        GVL_DataLogger.Seq := GVL_DataLogger.Seq + 1;
    END_IF
END_IF

IF (NOT GVL_NimServo.Enable) AND (NOT GVL_PD33.Enable) AND (NOT GVL_Vibration.Enable) AND GVL_Rs485Demo.Enable THEN
// --- EL6022 RS-485 demo loopback (Ch1 <-> Ch2) ---
// One-time init handshake (Ctrl bit2 / Status bit2)
IF NOT initCh1Done THEN
    GVL_EL6022_IO.EL6022_Ch1_Ctrl := GVL_EL6022_IO.EL6022_Ch1_Ctrl OR 16#0004;
    IF (GVL_EL6022_IO.EL6022_Ch1_Status AND 16#0004) <> 0 THEN
        GVL_EL6022_IO.EL6022_Ch1_Ctrl := GVL_EL6022_IO.EL6022_Ch1_Ctrl AND 16#FFFB;
        initCh1Done := TRUE;
    END_IF
END_IF

IF NOT initCh2Done THEN
    GVL_EL6022_IO.EL6022_Ch2_Ctrl := GVL_EL6022_IO.EL6022_Ch2_Ctrl OR 16#0004;
    IF (GVL_EL6022_IO.EL6022_Ch2_Status AND 16#0004) <> 0 THEN
        GVL_EL6022_IO.EL6022_Ch2_Ctrl := GVL_EL6022_IO.EL6022_Ch2_Ctrl AND 16#FFFB;
        initCh2Done := TRUE;
    END_IF
END_IF

// TX handshake: low byte bits: b0=TxReq, b1=RxAck, b2=InitReq, b3=SendContinuous, high byte = length
IF (GVL_Rs485Demo.TxBusy = FALSE) AND (GVL_Rs485Demo.TxSeq <> GVL_Rs485Demo.TxDoneSeq) THEN
    // Prepare control word for selected TX channel
    IF GVL_Rs485Demo.TxUseCh2 THEN
        // Copy TX payload
        GVL_EL6022_IO.EL6022_Ch2_DataOut := GVL_Rs485Demo.TxData;
        // Set length (high byte) and TxReq (bit0)
        GVL_EL6022_IO.EL6022_Ch2_Ctrl := (GVL_EL6022_IO.EL6022_Ch2_Ctrl AND 16#00FF) OR 16#0001 OR SHL(USINT_TO_WORD(GVL_Rs485Demo.TxLen), 8);
    ELSE
        GVL_EL6022_IO.EL6022_Ch1_DataOut := GVL_Rs485Demo.TxData;
        GVL_EL6022_IO.EL6022_Ch1_Ctrl := (GVL_EL6022_IO.EL6022_Ch1_Ctrl AND 16#00FF) OR 16#0001 OR SHL(USINT_TO_WORD(GVL_Rs485Demo.TxLen), 8);
    END_IF

    GVL_Rs485Demo.TxBusy := TRUE;
END_IF

// Observe Tx accepted on the selected channel (Status bit0)
IF GVL_Rs485Demo.TxBusy THEN
    IF GVL_Rs485Demo.TxUseCh2 THEN
        IF (GVL_EL6022_IO.EL6022_Ch2_Status AND 16#0001) <> 0 THEN
            // Clear TxReq bit after accepted
            GVL_EL6022_IO.EL6022_Ch2_Ctrl := GVL_EL6022_IO.EL6022_Ch2_Ctrl AND 16#00FE;
            GVL_Rs485Demo.TxDoneSeq := GVL_Rs485Demo.TxSeq;
            GVL_Rs485Demo.TxBusy := FALSE;
        END_IF
    ELSE
        IF (GVL_EL6022_IO.EL6022_Ch1_Status AND 16#0001) <> 0 THEN
            GVL_EL6022_IO.EL6022_Ch1_Ctrl := GVL_EL6022_IO.EL6022_Ch1_Ctrl AND 16#00FE;
            GVL_Rs485Demo.TxDoneSeq := GVL_Rs485Demo.TxSeq;
            GVL_Rs485Demo.TxBusy := FALSE;
        END_IF
    END_IF
END_IF

// RX handling: Status bit1=Receive request, high byte = input length
IF (GVL_EL6022_IO.EL6022_Ch1_Status AND 16#0002) <> 0 THEN
    GVL_Rs485Demo.RxFromCh2 := FALSE;
    GVL_Rs485Demo.RxStatus := GVL_EL6022_IO.EL6022_Ch1_Status;
    GVL_Rs485Demo.RxLen := WORD_TO_USINT(SHR(GVL_EL6022_IO.EL6022_Ch1_Status, 8));
    GVL_Rs485Demo.RxData := GVL_EL6022_IO.EL6022_Ch1_DataIn;
    GVL_Rs485Demo.RxSeq := GVL_Rs485Demo.RxSeq + 1;
    // Acknowledge receive (Ctrl bit1)
    GVL_EL6022_IO.EL6022_Ch1_Ctrl := GVL_EL6022_IO.EL6022_Ch1_Ctrl OR 16#0002;
ELSIF (GVL_EL6022_IO.EL6022_Ch2_Status AND 16#0002) <> 0 THEN
    GVL_Rs485Demo.RxFromCh2 := TRUE;
    GVL_Rs485Demo.RxStatus := GVL_EL6022_IO.EL6022_Ch2_Status;
    GVL_Rs485Demo.RxLen := WORD_TO_USINT(SHR(GVL_EL6022_IO.EL6022_Ch2_Status, 8));
    GVL_Rs485Demo.RxData := GVL_EL6022_IO.EL6022_Ch2_DataIn;
    GVL_Rs485Demo.RxSeq := GVL_Rs485Demo.RxSeq + 1;
    GVL_EL6022_IO.EL6022_Ch2_Ctrl := GVL_EL6022_IO.EL6022_Ch2_Ctrl OR 16#0002;
ELSE
    // Drop RxAck bits when no receive request pending
    GVL_EL6022_IO.EL6022_Ch1_Ctrl := GVL_EL6022_IO.EL6022_Ch1_Ctrl AND 16#FFFD;
    GVL_EL6022_IO.EL6022_Ch2_Ctrl := GVL_EL6022_IO.EL6022_Ch2_Ctrl AND 16#FFFD;
END_IF
END_IF

END_PROGRAM

// ---- POUs/FB_NimServo.TcPOU
FUNCTION_BLOCK FB_NimServo
VAR_INPUT
    Enable : BOOL;
    Channel : USINT;
    SlaveId : USINT;

    AutoSetCia402Mode : BOOL;
    DesiredMode : USINT; // 2=VM, 9=CSV
    PowerEnable : BOOL;
    TargetVelocity : DINT;
    WordSwap32 : BOOL;
    TestForceVelocityWrite : BOOL;
    ExtendedPoll : BOOL; // TRUE: poll extended diagnostics (more traffic)
    ApplyVmConfig : BOOL; // TRUE: write VM params (min/max/accel/decel) when PowerEnable=FALSE

    VmSpeedMinRpm : UDINT;
    VmSpeedMaxRpm : UDINT;
    VmAccelRpm : UDINT;
    VmAccelTimeS : UINT;
    VmDecelRpm : UDINT;
    VmDecelTimeS : UINT;

    CmdSeq : UDINT;
    Cmd : USINT; // 0=None, 1=FaultReset
END_VAR
VAR_OUTPUT
    CmdAckSeq : UDINT;
    Busy : BOOL;
    CommOk : BOOL;
    CommErrorCount : UDINT;
    LastErrorId : UDINT;

    ControlMode : USINT;
    ControlModeOk : BOOL;
    StatusWord : UINT;
    ControlWord : UINT;

    Cia402State : USINT;
    ErrorRegister : USINT;
    CurrentAlarm : USINT;

    DiSignals : UINT;
    DoSignals : UINT;
    DcBusVoltage : UINT;
    ModuleTemp : INT;

    Di1Func : USINT;
    Di1Logic : USINT;
    Di2Func : USINT;
    Di2Logic : USINT;
    Di3Func : USINT;
    Di3Logic : USINT;
    Di4Func : USINT;
    Di4Logic : USINT;
    Di5Func : USINT;
    Di5Logic : USINT;
    Di6Func : USINT;
    Di6Logic : USINT;
    Di7Func : USINT;
    Di7Logic : USINT;
    Di8Func : USINT;
    Di8Logic : USINT;
    Di9Func : USINT;
    Di9Logic : USINT;

    EnableDiIndex : USINT;
    EnableDiRequired : BOOL;
    EnableDiActive : BOOL;
    EnableDiOk : BOOL;

    DriveInternalState : USINT;
    FpgaSystemStatus : UINT;
    FpgaSystemFault : UINT;
    EncoderInternalFault : UINT;
    FaultRecord : UINT;
    AbsEncoderWord : UINT;

    ModeDisplay : USINT;
    ActualVelocity : DINT;
    ActualPosition : DINT;
    CurrentFeedback : INT;

    VmTargetSpeedRpm : INT;
    VmTargetSpeedEffRpm : INT;
    VmActualSpeedRpm : INT;

    VmCfgPendingOut : BOOL;
    VmCfgIndexOut : USINT;


    LastTxLen : USINT;
    LastTx : ARRAY [0..21] OF USINT;
    LastRxLen : USINT;
    LastRx : ARRAY [0..21] OF USINT;
END_VAR
VAR
    mb : FB_ModbusRtuMaster;
    mbReqHold : BOOL;
    mbFunc : USINT;
    mbAddr : UINT;
    mbQty : USINT;
    mbWbc : USINT;
    mbWData : ARRAY [0..21] OF USINT;

    op : USINT;
    step : USINT;

    desiredCtrl : UINT;
    faultResetPending : BOOL;
    cmdSeqLatched : UDINT;

    lastTargetVelocity : DINT;
    velWritePending : BOOL;

    vmCfgPending : BOOL;
    vmCfgStage : USINT; // 0=min/max, 1=accel/decel, 2=done
    vmCfgIndex : USINT; // 0..9 (single-register writes)
    vmStopPending : BOOL;
    lastVmSpeedMin : UDINT;
    lastVmSpeedMax : UDINT;
    lastVmAccel : UDINT;
    lastVmDecel : UDINT;
    lastVmAccelTimeS : UINT;
    lastVmDecelTimeS : UINT;

    lastDesiredMode : USINT;
    modeWritePending : BOOL;
    enablePrev : BOOL;
    powerEnablePrev : BOOL;
    forceCtrlWrite : BOOL;

    cfgDone : BOOL;
    cfgWritePending : BOOL;

    uTmp : UDINT;
    hi : UINT;
    lo : UINT;
    dw : DWORD;

    di1High : BOOL;
    di2High : BOOL;
    di3High : BOOL;
    di4High : BOOL;
    di5High : BOOL;
    di6High : BOOL;
    di7High : BOOL;
    di8High : BOOL;
    di9High : BOOL;
    diSelHigh : BOOL;

    iTmp : INT;

    tVmStartDelay : TON;
    driveStatePrev : USINT;
    applyVmConfigPrev : BOOL;
END_VAR

IF NOT Enable THEN
    Busy := FALSE;
    CommOk := FALSE;
    mbReqHold := FALSE;
    op := 0;
    step := 0;
    faultResetPending := FALSE;
    modeWritePending := FALSE;
    enablePrev := FALSE;
    powerEnablePrev := FALSE;
    forceCtrlWrite := FALSE;
    cfgDone := FALSE;
    cfgWritePending := FALSE;
    lastDesiredMode := 0;
    lastTargetVelocity := 0;
    lastVmSpeedMin := 0;
    lastVmSpeedMax := 0;
    lastVmAccel := 0;
    lastVmDecel := 0;
    lastVmAccelTimeS := 0;
    lastVmDecelTimeS := 0;

    Cia402State := 0;
    ErrorRegister := 0;
    CurrentAlarm := 0;
    DiSignals := 0;
    DoSignals := 0;
    DcBusVoltage := 0;
    ModuleTemp := 0;
    Di1Func := 0;
    Di1Logic := 0;
    Di2Func := 0;
    Di2Logic := 0;
    Di3Func := 0;
    Di3Logic := 0;
    Di4Func := 0;
    Di4Logic := 0;
    Di5Func := 0;
    Di5Logic := 0;
    Di6Func := 0;
    Di6Logic := 0;
    Di7Func := 0;
    Di7Logic := 0;
    Di8Func := 0;
    Di8Logic := 0;
    Di9Func := 0;
    Di9Logic := 0;
    EnableDiIndex := 0;
    EnableDiRequired := FALSE;
    EnableDiActive := FALSE;
    EnableDiOk := FALSE;
    DriveInternalState := 0;
    FpgaSystemStatus := 0;
    FpgaSystemFault := 0;
    EncoderInternalFault := 0;
    FaultRecord := 0;
    AbsEncoderWord := 0;

    VmTargetSpeedRpm := 0;
    VmTargetSpeedEffRpm := 0;
    VmActualSpeedRpm := 0;
    vmCfgPending := FALSE;
    vmCfgStage := 0;
    vmCfgIndex := 0;
    vmStopPending := FALSE;
    velWritePending := FALSE;
    ControlWord := 0;
    tVmStartDelay(IN := FALSE, PT := T#200ms);
    driveStatePrev := 0;
    applyVmConfigPrev := FALSE;
    RETURN;
END_IF

// VM start delay (align with SDK's post-power_on delay)
tVmStartDelay(IN := PowerEnable, PT := T#200ms);

IF Enable AND (NOT enablePrev) THEN
    // On enable rising edge: force a mode write at least once
    modeWritePending := TRUE;
    // Do not auto-write VM config on Enable; only apply when parameters are changed explicitly.
    vmCfgPending := FALSE;
    vmCfgStage := 0;
    vmCfgIndex := 0;
    lastVmSpeedMin := VmSpeedMinRpm;
    lastVmSpeedMax := VmSpeedMaxRpm;
    lastVmAccel := VmAccelRpm;
    lastVmDecel := VmDecelRpm;
    lastVmAccelTimeS := VmAccelTimeS;
    lastVmDecelTimeS := VmDecelTimeS;
    forceCtrlWrite := TRUE;
    velWritePending := TRUE;
END_IF
enablePrev := Enable;

// PowerEnable rising edge: re-assert controlword and speed (idempotent start)
IF PowerEnable AND (NOT powerEnablePrev) THEN
    forceCtrlWrite := TRUE;
    velWritePending := TRUE;
END_IF
// PowerEnable falling edge: in VM mode, command target speed = 0 once to ensure stop
IF (NOT PowerEnable) AND powerEnablePrev THEN
    IF DesiredMode = 2 THEN
        vmStopPending := TRUE;
    END_IF
END_IF
powerEnablePrev := PowerEnable;

IF DesiredMode <> lastDesiredMode THEN
    lastDesiredMode := DesiredMode;
    modeWritePending := TRUE;
END_IF

// Track target velocity change (for debug or for normal writes once comm works)
IF TargetVelocity <> lastTargetVelocity THEN
    lastTargetVelocity := TargetVelocity;
    // VM mode uses VM target speed register (H0382), so we should treat it as a pending write too.
    velWritePending := TRUE;
    IF TestForceVelocityWrite THEN
        velWritePending := TRUE;
    END_IF
END_IF

// Track VM parameter changes (only applied when DesiredMode=VM)
IF ApplyVmConfig THEN
    IF (VmSpeedMinRpm <> lastVmSpeedMin) OR (VmSpeedMaxRpm <> lastVmSpeedMax) OR (VmAccelRpm <> lastVmAccel) OR (VmDecelRpm <> lastVmDecel) OR (VmAccelTimeS <> lastVmAccelTimeS) OR (VmDecelTimeS <> lastVmDecelTimeS) THEN
        lastVmSpeedMin := VmSpeedMinRpm;
        lastVmSpeedMax := VmSpeedMaxRpm;
        lastVmAccel := VmAccelRpm;
        lastVmDecel := VmDecelRpm;
        lastVmAccelTimeS := VmAccelTimeS;
        lastVmDecelTimeS := VmDecelTimeS;
        vmCfgPending := TRUE;
        vmCfgStage := 0;
        vmCfgIndex := 0;
    END_IF
ELSE
    // When not applying config, keep last values in sync and clear any leftover pending state.
    lastVmSpeedMin := VmSpeedMinRpm;
    lastVmSpeedMax := VmSpeedMaxRpm;
    lastVmAccel := VmAccelRpm;
    lastVmDecel := VmDecelRpm;
    lastVmAccelTimeS := VmAccelTimeS;
    lastVmDecelTimeS := VmDecelTimeS;
    vmCfgPending := FALSE;
    vmCfgIndex := 0;
END_IF

// Rising edge: (re)apply current VM config on next idle slot (while PowerEnable=FALSE)
IF ApplyVmConfig AND (NOT applyVmConfigPrev) THEN
    vmCfgPending := TRUE;
    vmCfgIndex := 0;
END_IF
applyVmConfigPrev := ApplyVmConfig;

// Latch one-shot command
IF (CmdSeq <> CmdAckSeq) AND (NOT faultResetPending) THEN
    cmdSeqLatched := CmdSeq;
    IF Cmd = 1 THEN
        faultResetPending := TRUE;
    ELSE
        // unknown command: ack immediately
        CmdAckSeq := CmdSeq;
    END_IF
END_IF

// Drive Modbus master
mb(Enable := Enable,
   Channel := Channel,
   SlaveId := SlaveId,
   Req := mbReqHold,
   Func := mbFunc,
   Addr := mbAddr,
   Quantity := mbQty,
   WriteByteCount := mbWbc,
   WriteData := mbWData);
IF mb.Busy THEN
    // Request accepted by Modbus FB
    mbReqHold := FALSE;
END_IF

Busy := mb.Busy;

// Update debug frames (latch last non-empty frames)
IF mb.TxLen > 0 THEN
    LastTxLen := mb.TxLen;
    LastTx := mb.TxFrame;
END_IF

IF mb.RxLen > 0 THEN
    LastRxLen := mb.RxLen;
    LastRx := mb.RxFrame;
END_IF

IF mb.Error THEN
    CommOk := FALSE;
    CommErrorCount := CommErrorCount + 1;
    LastErrorId := mb.ErrorId;

    // Re-arm pending writes on error so we retry.
    IF op = 11 THEN
        cfgWritePending := TRUE;
    ELSIF op = 6 THEN
        modeWritePending := TRUE;
    ELSIF op = 8 THEN
        velWritePending := TRUE;
    ELSIF op = 25 THEN
        vmStopPending := TRUE;
    ELSIF op = 23 THEN
        IF ApplyVmConfig THEN
            vmCfgPending := TRUE;
        ELSE
            vmCfgPending := FALSE;
            vmCfgIndex := 0;
        END_IF
    END_IF

    op := 0;
    // stay on the same step when comm is down; allow pending debug writes to still be sent
END_IF

IF mb.Done THEN
    CommOk := TRUE;

    CASE op OF
    10: // ControlMode (I2002-1 / H00B1)
        ControlMode := WORD_TO_USINT(UINT_TO_WORD(mb.ReadRegs[0] AND 16#00FF));
        IF ControlMode = 0 THEN
            ControlModeOk := TRUE;
            cfgDone := TRUE;
        ELSE
            ControlModeOk := FALSE;
            cfgWritePending := TRUE;
            // Stay in preflight until mode is correct (or AutoSet disabled)
            IF NOT AutoSetCia402Mode THEN
                cfgDone := TRUE; // user will handle manually
            END_IF
        END_IF
    11: // Write ControlMode done (read back next)
        cfgDone := FALSE;
    1: // StatusWord
        StatusWord := mb.ReadRegs[0];
    22: // VM telemetry (I6042..I6044 / H0382..H0384)
        VmTargetSpeedRpm := WORD_TO_INT(UINT_TO_WORD(mb.ReadRegs[0]));
        VmTargetSpeedEffRpm := WORD_TO_INT(UINT_TO_WORD(mb.ReadRegs[1]));
        VmActualSpeedRpm := WORD_TO_INT(UINT_TO_WORD(mb.ReadRegs[2]));
    12: // DiSignals (I200B-5 / H01E2)
        DiSignals := mb.ReadRegs[0];
    18: // DoSignals (I200B-6 / H01E3)
        DoSignals := mb.ReadRegs[0];
    19: // Bus voltage & temp (I200B-21/22 / H01F7..H01F8)
        DcBusVoltage := mb.ReadRegs[0];
        ModuleTemp := WORD_TO_INT(UINT_TO_WORD(mb.ReadRegs[1]));
    13: // DriveInternalState (I200B-1 / H01DE)
        DriveInternalState := WORD_TO_USINT(UINT_TO_WORD(mb.ReadRegs[0] AND 16#00FF));
    17: // FPGA abs encoder + system status/fault (I200B-23..27 / H01F9..H01FD)
        AbsEncoderWord := mb.ReadRegs[0];
        FpgaSystemStatus := mb.ReadRegs[1];
        FpgaSystemFault := mb.ReadRegs[2];
        EncoderInternalFault := mb.ReadRegs[3];
        FaultRecord := mb.ReadRegs[4];
    14: // ErrorRegister (I1001 / H0000, low byte)
        ErrorRegister := WORD_TO_USINT(UINT_TO_WORD(mb.ReadRegs[0] AND 16#00FF));
    15: // CurrentAlarm (I1003-0 / H0001, low byte)
        CurrentAlarm := WORD_TO_USINT(UINT_TO_WORD(mb.ReadRegs[0] AND 16#00FF));
    2: // ModeDisplay (low byte)
        ModeDisplay := WORD_TO_USINT(UINT_TO_WORD(mb.ReadRegs[0] AND 16#00FF));
    3: // ActualVelocity (2 regs)
        hi := mb.ReadRegs[0];
        lo := mb.ReadRegs[1];
        IF WordSwap32 THEN
            hi := mb.ReadRegs[1];
            lo := mb.ReadRegs[0];
        END_IF
        uTmp := SHL(UINT_TO_UDINT(hi), 16) OR UINT_TO_UDINT(lo);
        dw := UDINT_TO_DWORD(uTmp);
        ActualVelocity := DWORD_TO_DINT(dw);
    4: // ActualPosition (2 regs)
        hi := mb.ReadRegs[0];
        lo := mb.ReadRegs[1];
        IF WordSwap32 THEN
            hi := mb.ReadRegs[1];
            lo := mb.ReadRegs[0];
        END_IF
        uTmp := SHL(UINT_TO_UDINT(hi), 16) OR UINT_TO_UDINT(lo);
        dw := UDINT_TO_DWORD(uTmp);
        ActualPosition := DWORD_TO_DINT(dw);
    5: // CurrentFeedback (16-bit signed)
        CurrentFeedback := WORD_TO_INT(UINT_TO_WORD(mb.ReadRegs[0]));
    16: // DI1..DI4 config (I2003-3..10 / H00D5..H00DC), low byte per register
        Di1Func := WORD_TO_USINT(UINT_TO_WORD(mb.ReadRegs[0] AND 16#00FF));
        Di1Logic := WORD_TO_USINT(UINT_TO_WORD(mb.ReadRegs[1] AND 16#00FF));
        Di2Func := WORD_TO_USINT(UINT_TO_WORD(mb.ReadRegs[2] AND 16#00FF));
        Di2Logic := WORD_TO_USINT(UINT_TO_WORD(mb.ReadRegs[3] AND 16#00FF));
        Di3Func := WORD_TO_USINT(UINT_TO_WORD(mb.ReadRegs[4] AND 16#00FF));
        Di3Logic := WORD_TO_USINT(UINT_TO_WORD(mb.ReadRegs[5] AND 16#00FF));
        Di4Func := WORD_TO_USINT(UINT_TO_WORD(mb.ReadRegs[6] AND 16#00FF));
        Di4Logic := WORD_TO_USINT(UINT_TO_WORD(mb.ReadRegs[7] AND 16#00FF));
    20: // DI5..DI8 config (I2003-11..18 / H00DD..H00E4), low byte per register
        Di5Func := WORD_TO_USINT(UINT_TO_WORD(mb.ReadRegs[0] AND 16#00FF));
        Di5Logic := WORD_TO_USINT(UINT_TO_WORD(mb.ReadRegs[1] AND 16#00FF));
        Di6Func := WORD_TO_USINT(UINT_TO_WORD(mb.ReadRegs[2] AND 16#00FF));
        Di6Logic := WORD_TO_USINT(UINT_TO_WORD(mb.ReadRegs[3] AND 16#00FF));
        Di7Func := WORD_TO_USINT(UINT_TO_WORD(mb.ReadRegs[4] AND 16#00FF));
        Di7Logic := WORD_TO_USINT(UINT_TO_WORD(mb.ReadRegs[5] AND 16#00FF));
        Di8Func := WORD_TO_USINT(UINT_TO_WORD(mb.ReadRegs[6] AND 16#00FF));
        Di8Logic := WORD_TO_USINT(UINT_TO_WORD(mb.ReadRegs[7] AND 16#00FF));
    21: // DI9 config (I2003-19..20 / H00E5..H00E6)
        Di9Func := WORD_TO_USINT(UINT_TO_WORD(mb.ReadRegs[0] AND 16#00FF));
        Di9Logic := WORD_TO_USINT(UINT_TO_WORD(mb.ReadRegs[1] AND 16#00FF));
    6: // WriteMode done
        ;
    7: // WriteControl done
        forceCtrlWrite := FALSE;
    8: // WriteTargetVel done
        ;
    25: // VM stop (write H0382=0) done
        vmStopPending := FALSE;
    23: // Write VM cfg single register done
        IF vmCfgIndex < 9 THEN
            vmCfgIndex := vmCfgIndex + 1;
            vmCfgPending := TRUE;
        ELSE
            vmCfgPending := FALSE;
        END_IF
    ELSE
        ;
    END_CASE

    op := 0;
    step := step + 1;
    IF step > 18 THEN
        step := 0;
    END_IF
END_IF

// expose VM config progress
VmCfgPendingOut := vmCfgPending;
VmCfgIndexOut := vmCfgIndex;

// If drive transitions from "not ready" to "ready/loop active", re-assert control and target speed once.
IF (driveStatePrev = 0) AND (DriveInternalState <> 0) THEN
    forceCtrlWrite := TRUE;
    velWritePending := TRUE;
END_IF
driveStatePrev := DriveInternalState;

// Derive CiA402 state (DS402)
IF (StatusWord AND 16#004F) = 16#0008 THEN
    Cia402State := 7; // Fault
ELSIF (StatusWord AND 16#004F) = 16#000F THEN
    Cia402State := 6; // Fault reaction active
ELSIF (StatusWord AND 16#006F) = 16#0027 THEN
    Cia402State := 5; // Operation enabled
ELSIF (StatusWord AND 16#006F) = 16#0023 THEN
    Cia402State := 4; // Switched on
ELSIF (StatusWord AND 16#006F) = 16#0021 THEN
    Cia402State := 3; // Ready to switch on
ELSIF (StatusWord AND 16#006F) = 16#0007 THEN
    Cia402State := 8; // Quick stop active
ELSIF (StatusWord AND 16#004F) = 16#0040 THEN
    Cia402State := 2; // Switch on disabled
ELSIF (StatusWord AND 16#004F) = 16#0000 THEN
    Cia402State := 1; // Not ready to switch on
ELSE
    Cia402State := 0; // Unknown
END_IF

// Derive DI enable status (based on DI1 settings)
di1High := (DiSignals AND 16#0001) <> 0;
di2High := (DiSignals AND 16#0002) <> 0;
di3High := (DiSignals AND 16#0004) <> 0;
di4High := (DiSignals AND 16#0008) <> 0;
di5High := (DiSignals AND 16#0010) <> 0;
di6High := (DiSignals AND 16#0020) <> 0;
di7High := (DiSignals AND 16#0040) <> 0;
di8High := (DiSignals AND 16#0080) <> 0;
di9High := (DiSignals AND 16#0100) <> 0;

EnableDiIndex := 0;
IF Di1Func = 1 THEN
    EnableDiIndex := 1;
ELSIF Di2Func = 1 THEN
    EnableDiIndex := 2;
ELSIF Di3Func = 1 THEN
    EnableDiIndex := 3;
ELSIF Di4Func = 1 THEN
    EnableDiIndex := 4;
ELSIF Di5Func = 1 THEN
    EnableDiIndex := 5;
ELSIF Di6Func = 1 THEN
    EnableDiIndex := 6;
ELSIF Di7Func = 1 THEN
    EnableDiIndex := 7;
ELSIF Di8Func = 1 THEN
    EnableDiIndex := 8;
ELSIF Di9Func = 1 THEN
    EnableDiIndex := 9;
END_IF
EnableDiRequired := EnableDiIndex <> 0;

diSelHigh := FALSE;
IF EnableDiIndex = 1 THEN
    diSelHigh := di1High;
ELSIF EnableDiIndex = 2 THEN
    diSelHigh := di2High;
ELSIF EnableDiIndex = 3 THEN
    diSelHigh := di3High;
ELSIF EnableDiIndex = 4 THEN
    diSelHigh := di4High;
ELSIF EnableDiIndex = 5 THEN
    diSelHigh := di5High;
ELSIF EnableDiIndex = 6 THEN
    diSelHigh := di6High;
ELSIF EnableDiIndex = 7 THEN
    diSelHigh := di7High;
ELSIF EnableDiIndex = 8 THEN
    diSelHigh := di8High;
ELSIF EnableDiIndex = 9 THEN
    diSelHigh := di9High;
END_IF

IF EnableDiRequired THEN
    // Logic selection value is stored per DI (0=low active, 1=high active)
    IF (EnableDiIndex = 1) AND (Di1Logic = 0) THEN
        EnableDiActive := NOT diSelHigh;
    ELSIF (EnableDiIndex = 1) AND (Di1Logic = 1) THEN
        EnableDiActive := diSelHigh;
    ELSIF (EnableDiIndex = 2) AND (Di2Logic = 0) THEN
        EnableDiActive := NOT diSelHigh;
    ELSIF (EnableDiIndex = 2) AND (Di2Logic = 1) THEN
        EnableDiActive := diSelHigh;
    ELSIF (EnableDiIndex = 3) AND (Di3Logic = 0) THEN
        EnableDiActive := NOT diSelHigh;
    ELSIF (EnableDiIndex = 3) AND (Di3Logic = 1) THEN
        EnableDiActive := diSelHigh;
    ELSIF (EnableDiIndex = 4) AND (Di4Logic = 0) THEN
        EnableDiActive := NOT diSelHigh;
    ELSIF (EnableDiIndex = 4) AND (Di4Logic = 1) THEN
        EnableDiActive := diSelHigh;
    ELSIF (EnableDiIndex = 5) AND (Di5Logic = 0) THEN
        EnableDiActive := NOT diSelHigh;
    ELSIF (EnableDiIndex = 5) AND (Di5Logic = 1) THEN
        EnableDiActive := diSelHigh;
    ELSIF (EnableDiIndex = 6) AND (Di6Logic = 0) THEN
        EnableDiActive := NOT diSelHigh;
    ELSIF (EnableDiIndex = 6) AND (Di6Logic = 1) THEN
        EnableDiActive := diSelHigh;
    ELSIF (EnableDiIndex = 7) AND (Di7Logic = 0) THEN
        EnableDiActive := NOT diSelHigh;
    ELSIF (EnableDiIndex = 7) AND (Di7Logic = 1) THEN
        EnableDiActive := diSelHigh;
    ELSIF (EnableDiIndex = 8) AND (Di8Logic = 0) THEN
        EnableDiActive := NOT diSelHigh;
    ELSIF (EnableDiIndex = 8) AND (Di8Logic = 1) THEN
        EnableDiActive := diSelHigh;
    ELSIF (EnableDiIndex = 9) AND (Di9Logic = 0) THEN
        EnableDiActive := NOT diSelHigh;
    ELSIF (EnableDiIndex = 9) AND (Di9Logic = 1) THEN
        EnableDiActive := diSelHigh;
    ELSE
        EnableDiActive := FALSE; // edge-based or unknown mode
    END_IF
ELSE
    EnableDiActive := TRUE;
END_IF
EnableDiOk := (NOT EnableDiRequired) OR EnableDiActive;

// Determine desired control word (simple CiA402 sequence)
desiredCtrl := 0;
IF faultResetPending THEN
    desiredCtrl := 16#0080;
ELSIF PowerEnable THEN
    // Fault?
    IF Cia402State = 7 THEN
        desiredCtrl := 16#0080;
    // VM mode: follow CiA402 state machine, then use 0x7F once op enabled (aligns with SDK behavior).
    ELSIF DesiredMode = 2 THEN
        IF Cia402State = 5 THEN
            desiredCtrl := 16#007F;
        ELSIF Cia402State = 4 THEN
            desiredCtrl := 16#000F;
        ELSIF Cia402State = 3 THEN
            desiredCtrl := 16#0007;
        ELSE
            // includes Switch on disabled / Not ready / Unknown
            desiredCtrl := 16#0006;
        END_IF
    ELSE
        // Other modes: standard CiA402 bring-up to operation enabled (0x0F)
        IF Cia402State = 5 THEN
            desiredCtrl := 16#000F; // operation enabled
        ELSIF Cia402State = 4 THEN
            desiredCtrl := 16#000F; // switch on -> enable operation
        ELSIF Cia402State = 3 THEN
            desiredCtrl := 16#0007; // ready -> switch on
        ELSE
            desiredCtrl := 16#0006; // shutdown
        END_IF
    END_IF
END_IF

// Schedule next Modbus transaction when idle
IF (NOT mb.Busy) AND (op = 0) AND mb.PortReady AND (NOT mbReqHold) THEN
    // Preflight: ensure control mode is CIA402 (I2002-1 / H00B1 = 0) if requested.
    IF NOT cfgDone THEN
        IF cfgWritePending AND AutoSetCia402Mode THEN
            mbFunc := 6;
            mbAddr := 16#00B1;
            mbQty := 1;
            mbWbc := 2;
            mbWData[0] := 0;
            mbWData[1] := 0;
            op := 11; // write control mode
            mbReqHold := TRUE;
            cfgWritePending := FALSE;
            RETURN;
        ELSE
            mbFunc := 3;
            mbAddr := 16#00B1;
            mbQty := 1;
            mbWbc := 0;
            op := 10; // read control mode
            mbReqHold := TRUE;
            RETURN;
        END_IF
    END_IF

    // VM stop on PowerEnable falling edge: write H0382 = 0 once (before changing controlword)
    IF vmStopPending AND (DesiredMode = 2) THEN
        mbFunc := 6;
        mbAddr := 16#0382;
        mbQty := 1;
        mbWbc := 2;
        mbWData[0] := 0;
        mbWData[1] := 0;
        op := 25;
        mbReqHold := TRUE;
        RETURN;
    END_IF

    // ControlWord has priority over speed writes (improves repeatability on re-start)
    IF (ControlWord <> desiredCtrl) OR forceCtrlWrite THEN
        ControlWord := desiredCtrl;
        mbFunc := 6;
        mbAddr := 16#0380;
        mbQty := 1;
        mbWbc := 2;
        mbWData[0] := WORD_TO_USINT(SHR(UINT_TO_WORD(ControlWord), 8));
        mbWData[1] := WORD_TO_USINT(UINT_TO_WORD(ControlWord) AND 16#00FF);
        op := 7;
        mbReqHold := TRUE;
        // clear fault reset after one write
        IF faultResetPending THEN
            faultResetPending := FALSE;
            CmdAckSeq := cmdSeqLatched;
        END_IF
        RETURN;
    END_IF

    // Debug: force a 60FF write when requested, even without OP enabled / without prior successful reads.
    IF velWritePending THEN
        IF DesiredMode = 2 THEN
            // Only send VM target speed when PowerEnable is asserted and after a short start delay.
            // Important: do NOT block the rest of the polling/state-machine when preconditions are not met yet.
            // Otherwise, writing TargetVelocity "too early" can starve StatusWord reads and prevent reaching OP enabled.
            IF (NOT PowerEnable) OR (NOT tVmStartDelay.Q) OR (Cia402State <> 5) THEN
                // keep pending; try again later
            ELSE

            // VM mode uses I6042 (H0382) "VM模式的目标速度", 16-bit signed rpm.
            iTmp := DINT_TO_INT(TargetVelocity);
            // Clamp to Modbus.db limits (-6000..6000 rpm) to avoid overflow/undefined behavior.
            IF iTmp > INT#6000 THEN
                iTmp := INT#6000;
            ELSIF iTmp < INT#-6000 THEN
                iTmp := INT#-6000;
            END_IF
            mbFunc := 6;
            mbAddr := 16#0382;
            mbQty := 1;
            mbWbc := 2;
            mbWData[0] := WORD_TO_USINT(SHR(INT_TO_WORD(iTmp), 8));
            mbWData[1] := WORD_TO_USINT(INT_TO_WORD(iTmp) AND 16#00FF);
            op := 8;
            mbReqHold := TRUE;
            velWritePending := FALSE;
            RETURN;
            END_IF
        ELSE
            // CSV (and others): use 60FF (H0448) 32-bit once OP enabled, unless forced.
            // Same as VM: never block the rest of the polling/state-machine when preconditions are not met yet.
            IF (NOT TestForceVelocityWrite) AND (NOT (PowerEnable AND (Cia402State = 5))) THEN
                // keep pending until drive is enabled
            ELSE

            dw := DINT_TO_DWORD(TargetVelocity);
            uTmp := DWORD_TO_UDINT(dw);
            hi := UDINT_TO_UINT(SHR(uTmp, 16));
            lo := UDINT_TO_UINT(uTmp AND 16#0000FFFF);

            mbFunc := 16;
            mbAddr := 16#0448;
            mbQty := 2;
            mbWbc := 4;

            IF WordSwap32 THEN
                // low word first
                mbWData[0] := WORD_TO_USINT(SHR(UINT_TO_WORD(lo), 8));
                mbWData[1] := WORD_TO_USINT(UINT_TO_WORD(lo) AND 16#00FF);
                mbWData[2] := WORD_TO_USINT(SHR(UINT_TO_WORD(hi), 8));
                mbWData[3] := WORD_TO_USINT(UINT_TO_WORD(hi) AND 16#00FF);
            ELSE
                // high word first
                mbWData[0] := WORD_TO_USINT(SHR(UINT_TO_WORD(hi), 8));
                mbWData[1] := WORD_TO_USINT(UINT_TO_WORD(hi) AND 16#00FF);
                mbWData[2] := WORD_TO_USINT(SHR(UINT_TO_WORD(lo), 8));
                mbWData[3] := WORD_TO_USINT(UINT_TO_WORD(lo) AND 16#00FF);
            END_IF

            op := 8;
            mbReqHold := TRUE;
            velWritePending := FALSE;
            RETURN;
            END_IF
        END_IF
    END_IF

    CASE step OF
    0: // Read StatusWord (6041 = H0381)
        mbFunc := 3;
        mbAddr := 16#0381;
        mbQty := 1;
        mbWbc := 0;
        op := 1;
        mbReqHold := TRUE;

    1: // Read DiSignals (I200B-5 = H01E2)
        IF ExtendedPoll THEN
            mbFunc := 3;
            mbAddr := 16#01E2;
            mbQty := 1;
            mbWbc := 0;
            op := 12;
            mbReqHold := TRUE;
        ELSE
            step := 17;
        END_IF

    2: // Read DoSignals (I200B-6 = H01E3)
        IF ExtendedPoll THEN
            mbFunc := 3;
            mbAddr := 16#01E3;
            mbQty := 1;
            mbWbc := 0;
            op := 18;
            mbReqHold := TRUE;
        ELSE
            step := 3;
        END_IF

    3: // Read Bus voltage & temp (I200B-21/22 = H01F7..H01F8)
        IF ExtendedPoll THEN
            mbFunc := 3;
            mbAddr := 16#01F7;
            mbQty := 2;
            mbWbc := 0;
            op := 19;
            mbReqHold := TRUE;
        ELSE
            step := 17;
        END_IF

    4: // Read DriveInternalState (I200B-1 = H01DE)
        IF ExtendedPoll THEN
            mbFunc := 3;
            mbAddr := 16#01DE;
            mbQty := 1;
            mbWbc := 0;
            op := 13;
            mbReqHold := TRUE;
        ELSE
            step := 17;
        END_IF

    5: // Read FPGA absolute encoder & system status/fault (I200B-23..27 = H01F9..H01FD)
        IF ExtendedPoll THEN
            mbFunc := 3;
            mbAddr := 16#01F9;
            mbQty := 5;
            mbWbc := 0;
            op := 17;
            mbReqHold := TRUE;
        ELSE
            step := 6;
        END_IF

    6: // Read ErrorRegister (I1001 = H0000)
        IF ExtendedPoll THEN
            mbFunc := 3;
            mbAddr := 16#0000;
            mbQty := 1;
            mbWbc := 0;
            op := 14;
            mbReqHold := TRUE;
        ELSE
            step := 17;
        END_IF

    7: // Read CurrentAlarm (I1003-0 = H0001)
        IF ExtendedPoll THEN
            mbFunc := 3;
            mbAddr := 16#0001;
            mbQty := 1;
            mbWbc := 0;
            op := 15;
            mbReqHold := TRUE;
        ELSE
            step := 17;
        END_IF

    8: // Read ModeDisplay (6061 = H03C3)
        IF ExtendedPoll THEN
            mbFunc := 3;
            mbAddr := 16#03C3;
            mbQty := 1;
            mbWbc := 0;
            op := 2;
            mbReqHold := TRUE;
        ELSE
            step := 17;
        END_IF

    9: // Read ActualVelocity (606C = H03D5, 2 regs)
        IF ExtendedPoll THEN
            mbFunc := 3;
            mbAddr := 16#03D5;
            mbQty := 2;
            mbWbc := 0;
            op := 3;
            mbReqHold := TRUE;
        ELSE
            step := 10;
        END_IF

    10: // Read ActualPosition (6064 = H03C8, 2 regs)
        IF ExtendedPoll THEN
            mbFunc := 3;
            mbAddr := 16#03C8;
            mbQty := 2;
            mbWbc := 0;
            op := 4;
            mbReqHold := TRUE;
        ELSE
            step := 11;
        END_IF

    11: // Read CurrentFeedback (6078 = H03E4)
        IF ExtendedPoll THEN
            mbFunc := 3;
            mbAddr := 16#03E4;
            mbQty := 1;
            mbWbc := 0;
            op := 5;
            mbReqHold := TRUE;
        ELSE
            step := 15;
        END_IF

    12: // Read DI1..DI4 config (I2003-3..10 = H00D5..H00DC)
        IF ExtendedPoll THEN
            mbFunc := 3;
            mbAddr := 16#00D5;
            mbQty := 8;
            mbWbc := 0;
            op := 16;
            mbReqHold := TRUE;
        ELSE
            step := 17;
        END_IF

    13: // Read DI5..DI8 config (I2003-11..18 = H00DD..H00E4)
        IF ExtendedPoll THEN
            mbFunc := 3;
            mbAddr := 16#00DD;
            mbQty := 8;
            mbWbc := 0;
            op := 20;
            mbReqHold := TRUE;
        ELSE
            step := 14;
        END_IF

    14: // Read DI9 config (I2003-19..20 = H00E5..H00E6)
        IF ExtendedPoll THEN
            mbFunc := 3;
            mbAddr := 16#00E5;
            mbQty := 2;
            mbWbc := 0;
            op := 21;
            mbReqHold := TRUE;
        ELSE
            step := 15;
        END_IF

    15: // VM config writes (only in VM mode)
        // Use single-register writes (0x06) for maximum device compatibility.
        // Also keep it before PowerEnable (aligns with SDK: power_off -> set params -> power_on).
        IF ApplyVmConfig AND vmCfgPending AND (DesiredMode = 2) AND (NOT PowerEnable) THEN
            mbFunc := 6;
            mbQty := 1;
            mbWbc := 2;

            CASE vmCfgIndex OF
            0: // H0385 min speed (hi word)
                uTmp := VmSpeedMinRpm;
                hi := UDINT_TO_UINT(SHR(uTmp, 16));
                mbAddr := 16#0385;
                mbWData[0] := WORD_TO_USINT(SHR(UINT_TO_WORD(hi), 8));
                mbWData[1] := WORD_TO_USINT(UINT_TO_WORD(hi) AND 16#00FF);
            1: // H0386 min speed (lo word)
                uTmp := VmSpeedMinRpm;
                lo := UDINT_TO_UINT(uTmp AND 16#0000FFFF);
                mbAddr := 16#0386;
                mbWData[0] := WORD_TO_USINT(SHR(UINT_TO_WORD(lo), 8));
                mbWData[1] := WORD_TO_USINT(UINT_TO_WORD(lo) AND 16#00FF);
            2: // H0387 max speed (hi word)
                uTmp := VmSpeedMaxRpm;
                hi := UDINT_TO_UINT(SHR(uTmp, 16));
                mbAddr := 16#0387;
                mbWData[0] := WORD_TO_USINT(SHR(UINT_TO_WORD(hi), 8));
                mbWData[1] := WORD_TO_USINT(UINT_TO_WORD(hi) AND 16#00FF);
            3: // H0388 max speed (lo word)
                uTmp := VmSpeedMaxRpm;
                lo := UDINT_TO_UINT(uTmp AND 16#0000FFFF);
                mbAddr := 16#0388;
                mbWData[0] := WORD_TO_USINT(SHR(UINT_TO_WORD(lo), 8));
                mbWData[1] := WORD_TO_USINT(UINT_TO_WORD(lo) AND 16#00FF);
            4: // H0389 accel (hi word)
                uTmp := VmAccelRpm;
                hi := UDINT_TO_UINT(SHR(uTmp, 16));
                mbAddr := 16#0389;
                mbWData[0] := WORD_TO_USINT(SHR(UINT_TO_WORD(hi), 8));
                mbWData[1] := WORD_TO_USINT(UINT_TO_WORD(hi) AND 16#00FF);
            5: // H038A accel (lo word)
                uTmp := VmAccelRpm;
                lo := UDINT_TO_UINT(uTmp AND 16#0000FFFF);
                mbAddr := 16#038A;
                mbWData[0] := WORD_TO_USINT(SHR(UINT_TO_WORD(lo), 8));
                mbWData[1] := WORD_TO_USINT(UINT_TO_WORD(lo) AND 16#00FF);
            6: // H038B accel time (seconds)
                mbAddr := 16#038B;
                mbWData[0] := WORD_TO_USINT(SHR(UINT_TO_WORD(VmAccelTimeS), 8));
                mbWData[1] := WORD_TO_USINT(UINT_TO_WORD(VmAccelTimeS) AND 16#00FF);
            7: // H038C decel (hi word)
                uTmp := VmDecelRpm;
                hi := UDINT_TO_UINT(SHR(uTmp, 16));
                mbAddr := 16#038C;
                mbWData[0] := WORD_TO_USINT(SHR(UINT_TO_WORD(hi), 8));
                mbWData[1] := WORD_TO_USINT(UINT_TO_WORD(hi) AND 16#00FF);
            8: // H038D decel (lo word)
                uTmp := VmDecelRpm;
                lo := UDINT_TO_UINT(uTmp AND 16#0000FFFF);
                mbAddr := 16#038D;
                mbWData[0] := WORD_TO_USINT(SHR(UINT_TO_WORD(lo), 8));
                mbWData[1] := WORD_TO_USINT(UINT_TO_WORD(lo) AND 16#00FF);
            ELSE // 9: H038E decel time (seconds)
                mbAddr := 16#038E;
                mbWData[0] := WORD_TO_USINT(SHR(UINT_TO_WORD(VmDecelTimeS), 8));
                mbWData[1] := WORD_TO_USINT(UINT_TO_WORD(VmDecelTimeS) AND 16#00FF);
            END_CASE

            op := 23;
            mbReqHold := TRUE;
            vmCfgPending := FALSE;
            RETURN;
        END_IF
        step := 16;

    16: // Write DesiredMode (6060 = H03C2) if needed
        IF modeWritePending AND ((DesiredMode = 2) OR (DesiredMode = 9)) THEN
            mbFunc := 6;
            mbAddr := 16#03C2;
            mbQty := 1;
            mbWbc := 2;
            mbWData[0] := 0;
            mbWData[1] := DesiredMode;
            op := 6;
            mbReqHold := TRUE;
            modeWritePending := FALSE;
            RETURN;
        END_IF
        step := 17;

    17: // Read VM telemetry (H0382..H0384), useful even when not ready
        mbFunc := 3;
        mbAddr := 16#0382;
        mbQty := 3;
        mbWbc := 0;
        op := 22;
        mbReqHold := TRUE;

    18: // (no-op; controlword handled in priority section above)
        step := 0;

    // Note: target speed writes are handled via velWritePending (H0382 for VM, 60FF for CSV).
    ELSE
        step := 0;
    END_CASE
END_IF

END_FUNCTION_BLOCK

// ---- POUs/FB_ModbusRtuMaster.TcPOU
FUNCTION_BLOCK FB_ModbusRtuMaster
VAR_INPUT
    Enable : BOOL;
    Channel : USINT; // 1 or 2
    SlaveId : USINT; // 1..247

    Req : BOOL;      // start a transaction when TRUE in IDLE
    Func : USINT;    // 3=Read Holding Registers, 6=Write Single Register, 16=Write Multiple Registers
    Addr : UINT;     // start address
    Quantity : USINT; // register count (read or write)

    WriteByteCount : USINT; // for 0x06 (2) or 0x10 (Quantity*2)
    WriteData : ARRAY [0..21] OF USINT; // big-endian per register

    Timeout : TIME := T#200ms;
    MinGap : TIME := T#20ms; // minimum silent time between Modbus frames (aligns with SDK PDOIntervalMS=20ms)
END_VAR
VAR_OUTPUT
    PortReady : BOOL;
    Busy : BOOL;
    Done : BOOL;
    Error : BOOL;
    ErrorId : UDINT;
    ExceptionCode : USINT;

    RxDiscardCount : UDINT;
    LastDiscardId : UDINT;

    ReadRegCount : USINT;
    ReadRegs : ARRAY [0..7] OF UINT;

    TxLen : USINT;
    TxFrame : ARRAY [0..21] OF USINT;
    RxLen : USINT;
    RxFrame : ARRAY [0..21] OF USINT;
END_VAR
VAR
    fbPort : FB_EL6022_Port;

    reqPrev : BOOL;
    reqEdge : BOOL;

    state : USINT;
    opFunc : USINT;
    opAddr : UINT;
    opQty : USINT;
    opWbc : USINT;
    opWData : ARRAY [0..21] OF USINT;

    txStart : BOOL;
    txStartPrev : BOOL;

    rxBuf : ARRAY [0..21] OF USINT;
    rxBufLen : USINT;

    tTimeout : TON;

    i : USINT;
    crc : WORD;
    rxCrc : WORD;
    calcCrc : WORD;

    expectedLen : USINT;
    byteCount : USINT;
    regCount : USINT;
    wbcExpected : USINT;

    gapActive : BOOL;
    tGap : TON;
END_VAR

Done := FALSE;
Error := FALSE;
ExceptionCode := 0;

// Backward compatible: keep the edge vars, but do not require a rising edge.
reqEdge := Req AND NOT reqPrev;
reqPrev := Req;

// Keep port running
fbPort(Enable := Enable, Channel := Channel, TxStart := txStart, TxLen := TxLen, TxData := TxFrame);
PortReady := fbPort.Ready;

// Minimum silent gap between transactions (prevents back-to-back frames that some devices dislike).
IF NOT Enable THEN
    gapActive := FALSE;
END_IF
tGap(IN := gapActive, PT := MinGap);
IF tGap.Q THEN
    gapActive := FALSE;
END_IF

// latch RX from port when available
IF fbPort.RxNew THEN
    rxBuf := fbPort.RxData;
    rxBufLen := fbPort.RxLen;
END_IF

// Timeout timer active only in WAIT_RX state
tTimeout(IN := (state = 40) AND Busy, PT := Timeout);

CASE state OF
0: // IDLE
    Busy := FALSE;
    ErrorId := 0;
    ReadRegCount := 0;
    // keep RxDiscardCount/LastDiscardId across cycles (diagnostics)
    rxBufLen := 0;
    RxLen := 0;
    TxLen := 0;
    txStart := FALSE;

    IF Req AND (NOT gapActive) THEN
        opFunc := Func;
        opAddr := Addr;
        opQty := Quantity;
        opWbc := WriteByteCount;
        opWData := WriteData;
        state := 10;
    END_IF

10: // WAIT_PORT_READY
    Busy := TRUE;
    txStart := FALSE;
    IF NOT Enable THEN
        state := 0;
    ELSIF PortReady THEN
        state := 20;
    END_IF

20: // BUILD + TX_START
    // Clear any previously latched RX for this new transaction
    rxBufLen := 0;

    // Build frame into TxFrame
    FOR i := 0 TO 21 DO
        TxFrame[i] := 0;
    END_FOR

    TxFrame[0] := SlaveId;
    TxFrame[1] := opFunc;
    TxFrame[2] := WORD_TO_USINT(SHR(UINT_TO_WORD(opAddr), 8));
    TxFrame[3] := WORD_TO_USINT(UINT_TO_WORD(opAddr) AND 16#00FF);
    TxFrame[4] := WORD_TO_USINT(SHR(USINT_TO_WORD(opQty), 8));
    TxFrame[5] := opQty;

    IF opFunc = 16 THEN
        // Safety: EL6022 data length is 22 bytes, TxFrame is [0..21].
        // Modbus 0x10 frame length = 7 + byteCount + 2, so byteCount must be <= 13 (and even).
        wbcExpected := opQty + opQty; // opQty * 2
        IF (opWbc = 0) OR (opWbc <> wbcExpected) OR (opWbc > 12) THEN
            Error := TRUE;
            ErrorId := 16#00010008; // invalid write byte count / frame too long
            Busy := FALSE;
            state := 70;
            RETURN;
        END_IF

        // Write multiple registers (0x10):
        // [6]=byteCount, [7..]=data bytes (big-endian per register)
        TxFrame[6] := opWbc;
        IF opWbc > 0 THEN
            FOR i := 0 TO opWbc - 1 DO
                TxFrame[7 + i] := opWData[i];
            END_FOR
        END_IF
        TxLen := 7 + opWbc + 2;
    ELSIF opFunc = 6 THEN
        // Write single register: WriteData[0..1] are hi/lo bytes
        TxFrame[4] := opWData[0];
        TxFrame[5] := opWData[1];
        TxLen := 8;
    ELSE
        // Read holding registers (0x03)
        opFunc := 3;
        TxFrame[1] := opFunc;
        TxLen := 8;
    END_IF

    // CRC (low byte first)
    crc := F_ModbusCrc16(TxFrame, TxLen - 2);
    TxFrame[TxLen - 2] := WORD_TO_USINT(crc AND 16#00FF);
    TxFrame[TxLen - 1] := WORD_TO_USINT(SHR(crc, 8));

    // start TX (one-cycle pulse)
    txStart := TRUE;
    state := 30;

30: // WAIT_TX_DONE
    // drop TX start pulse after one cycle
    txStart := FALSE;
    IF fbPort.TxDone THEN
        state := 40;
    END_IF

40: // WAIT_RX
    IF tTimeout.Q THEN
        Error := TRUE;
        ErrorId := 16#00010001; // timeout
        Busy := FALSE;
        state := 70;
    ELSIF rxBufLen > 0 THEN
        state := 50;
    END_IF

50: // PARSE
    // copy for debug output
    RxFrame := rxBuf;
    RxLen := rxBufLen;

    IF rxBufLen < 5 THEN
        // Some devices/interfaces may occasionally report a short/garbled frame.
        // Discard and keep waiting for a valid response within the same transaction timeout.
        RxDiscardCount := RxDiscardCount + 1;
        LastDiscardId := 16#00020002; // discard: short frame
        rxBufLen := 0;
        state := 40;
        RETURN;
    END_IF

    // CRC check
    rxCrc := USINT_TO_WORD(rxBuf[rxBufLen - 2]) OR SHL(USINT_TO_WORD(rxBuf[rxBufLen - 1]), 8);
    calcCrc := F_ModbusCrc16(rxBuf, rxBufLen - 2);
    IF rxCrc <> calcCrc THEN
        RxDiscardCount := RxDiscardCount + 1;
        LastDiscardId := 16#00020003; // discard: crc mismatch
        rxBufLen := 0;
        state := 40;
        RETURN;
    END_IF

    // Basic header check
    IF rxBuf[0] <> SlaveId THEN
        RxDiscardCount := RxDiscardCount + 1;
        LastDiscardId := 16#00020004; // discard: wrong slave id
        rxBufLen := 0;
        state := 40;
        RETURN;
    END_IF

    // Exception response
    IF rxBuf[1] = (opFunc + 16#80) THEN
        ExceptionCode := rxBuf[2];
        Error := TRUE;
        ErrorId := 16#00010005; // exception
        Busy := FALSE;
        state := 70;
        RETURN;
    END_IF

    // Expected responses
    IF opFunc = 3 THEN
        byteCount := rxBuf[2];
        expectedLen := 5 + byteCount;
        IF rxBufLen <> expectedLen THEN
            RxDiscardCount := RxDiscardCount + 1;
            LastDiscardId := 16#00020006; // discard: length mismatch
            rxBufLen := 0;
            state := 40;
            RETURN;
        END_IF

        regCount := byteCount / 2;
        IF regCount > 8 THEN
            regCount := 8;
        END_IF
        ReadRegCount := regCount;
        FOR i := 0 TO regCount - 1 DO
            ReadRegs[i] := SHL(USINT_TO_UINT(rxBuf[3 + (2 * i)]), 8) OR USINT_TO_UINT(rxBuf[4 + (2 * i)]);
        END_FOR
    ELSE
        // Write responses are fixed 8 bytes
        IF rxBufLen <> 8 THEN
            RxDiscardCount := RxDiscardCount + 1;
            LastDiscardId := 16#00020007; // discard: write response length mismatch
            rxBufLen := 0;
            state := 40;
            RETURN;
        END_IF
    END_IF

    Done := TRUE;
    Busy := FALSE;
    gapActive := TRUE;
    state := 60;

60: // DONE (one cycle)
    state := 0;

70: // ERROR (one cycle)
    gapActive := TRUE;
    state := 0;

ELSE
    state := 0;
END_CASE

END_FUNCTION_BLOCK

// ---- POUs/FB_EL6022_Port.TcPOU
FUNCTION_BLOCK FB_EL6022_Port
VAR_INPUT
    Enable : BOOL;
    Channel : USINT; // 1 or 2

    TxStart : BOOL;
    TxLen : USINT; // 0..22
    TxData : ARRAY [0..21] OF USINT;
END_VAR
VAR_OUTPUT
    Ready : BOOL;

    TxBusy : BOOL;
    TxDone : BOOL;

    RxNew : BOOL;
    RxLen : USINT;
    RxData : ARRAY [0..21] OF USINT;

    LastStatus : WORD;
    LastCtrl : WORD;
END_VAR
VAR
    txStartPrev : BOOL;
    rxLatched : BOOL;

    status : WORD;
    ctrl : WORD;
END_VAR

TxDone := FALSE;
RxNew := FALSE;

IF NOT Enable THEN
    Ready := FALSE;
    TxBusy := FALSE;
    rxLatched := FALSE;
    txStartPrev := TxStart;
    RETURN;
END_IF

// Select channel
IF Channel = 2 THEN
    status := GVL_EL6022_IO.EL6022_Ch2_Status;
    ctrl := GVL_EL6022_IO.EL6022_Ch2_Ctrl;
ELSE
    status := GVL_EL6022_IO.EL6022_Ch1_Status;
    ctrl := GVL_EL6022_IO.EL6022_Ch1_Ctrl;
END_IF

// One-time init handshake (Ctrl bit2 / Status bit2)
IF NOT Ready THEN
    ctrl := ctrl OR 16#0004;
    IF (status AND 16#0004) <> 0 THEN
        ctrl := ctrl AND 16#FFFB;
        Ready := TRUE;
    END_IF
END_IF

// TX edge detect
IF (TxStart AND NOT txStartPrev) AND Ready AND (NOT TxBusy) THEN
    TxBusy := TRUE;

    IF Channel = 2 THEN
        GVL_EL6022_IO.EL6022_Ch2_DataOut := TxData;
        ctrl := (ctrl AND 16#00FF) OR 16#0001 OR SHL(USINT_TO_WORD(TxLen), 8);
    ELSE
        GVL_EL6022_IO.EL6022_Ch1_DataOut := TxData;
        ctrl := (ctrl AND 16#00FF) OR 16#0001 OR SHL(USINT_TO_WORD(TxLen), 8);
    END_IF
END_IF
txStartPrev := TxStart;

// TX accepted (Status bit0)
IF TxBusy THEN
    IF (status AND 16#0001) <> 0 THEN
        ctrl := ctrl AND 16#00FE; // clear TxReq and TX length after accepted
        TxBusy := FALSE;
        TxDone := TRUE;
    END_IF
END_IF

// RX handling (Status bit1), high byte = input length
IF (status AND 16#0002) <> 0 THEN
    RxLen := WORD_TO_USINT(SHR(status, 8));
    IF NOT rxLatched THEN
        IF Channel = 2 THEN
            RxData := GVL_EL6022_IO.EL6022_Ch2_DataIn;
        ELSE
            RxData := GVL_EL6022_IO.EL6022_Ch1_DataIn;
        END_IF
        RxNew := TRUE;
        rxLatched := TRUE;
    END_IF

    ctrl := ctrl OR 16#0002; // RxAck (bit1)
ELSE
    rxLatched := FALSE;
    ctrl := ctrl AND 16#FFFD; // clear RxAck
END_IF

// Write back ctrl to selected channel
IF Channel = 2 THEN
    GVL_EL6022_IO.EL6022_Ch2_Ctrl := ctrl;
ELSE
    GVL_EL6022_IO.EL6022_Ch1_Ctrl := ctrl;
END_IF

LastStatus := status;
LastCtrl := ctrl;

END_FUNCTION_BLOCK

// ---- POUs/F_ModbusCrc16.TcPOU
FUNCTION F_ModbusCrc16 : WORD
VAR_INPUT
    Data : ARRAY [0..21] OF USINT;
    Len : USINT;
END_VAR
VAR
    crc : WORD;
    i : USINT;
    j : USINT;
END_VAR

crc := 16#FFFF;

IF Len = 0 THEN
    F_ModbusCrc16 := crc;
    RETURN;
END_IF

FOR i := 0 TO Len - 1 DO
    crc := crc XOR USINT_TO_WORD(Data[i]);

    FOR j := 0 TO 7 DO
        IF (crc AND 16#0001) <> 0 THEN
            crc := SHR(crc, 1);
            crc := crc XOR 16#A001;
        ELSE
            crc := SHR(crc, 1);
        END_IF
    END_FOR
END_FOR

F_ModbusCrc16 := crc;

END_FUNCTION

// ---- POUs/FB_PD33.TcPOU
FUNCTION_BLOCK FB_PD33
VAR_INPUT
    Enable : BOOL;
    Channel : USINT; // 1 or 2
    SlaveId : USINT; // 1..247
    WordSwap32 : BOOL; // TRUE: low word first (matches PD33 manual examples)
    UseDisplayRegister3B : BOOL; // reserved: PD33 now uses passive full-speed output parsing

    CmdSeq : UDINT;
    Cmd : USINT; // reserved in passive mode
END_VAR
VAR_OUTPUT
    CmdAckSeq : UDINT;
    Busy : BOOL;

    PortReady : BOOL;
    CommOk : BOOL;
    CommErrorCount : UDINT;
    LastErrorId : UDINT;
    ExceptionCode : USINT;
    RxDiscardCount : UDINT;
    LastDiscardId : UDINT;

    AbsRaw : DINT;
    RelRaw : DINT;
    AbsMm : LREAL;
    RelMm : LREAL;
    ZeroWord : UINT;

    LastTxLen : USINT;
    LastTx : ARRAY [0..21] OF USINT;
    LastRxLen : USINT;
    LastRx : ARRAY [0..21] OF USINT;
END_VAR
VAR
    fbPort : FB_EL6022_Port;
    txData : ARRAY [0..21] OF USINT;
    rx : ARRAY [0..21] OF USINT;
    rxLen : USINT;
    crcRx : WORD;
    crcCalc : WORD;
    low : UINT;
    high : UINT;
    uTmp : UDINT;
    dw : DWORD;
    i : USINT;
END_VAR

IF NOT Enable THEN
    fbPort(Enable := FALSE, Channel := Channel, TxStart := FALSE, TxLen := 0, TxData := txData);

    Busy := FALSE;
    PortReady := FALSE;
    CommOk := FALSE;
    AbsRaw := 0;
    RelRaw := 0;
    AbsMm := 0.0;
    RelMm := 0.0;
    ZeroWord := 0;
    LastTxLen := 0;
    LastRxLen := 0;
    LastErrorId := 0;
    ExceptionCode := 0;
    RxDiscardCount := 0;
    LastDiscardId := 0;
    RETURN;
END_IF

// Passive mode: PD33 is configured for full-speed active output.
// The PLC only initializes/acknowledges the EL6022 channel and parses received frames.
fbPort(Enable := TRUE, Channel := Channel, TxStart := FALSE, TxLen := 0, TxData := txData);

Busy := FALSE;
PortReady := fbPort.Ready;
ExceptionCode := 0;
LastTxLen := 0;

IF CmdSeq <> CmdAckSeq THEN
    // Active zero/cancel writes are intentionally disabled while the sensor is in full-speed output mode.
    CmdAckSeq := CmdSeq;
END_IF

IF fbPort.RxNew THEN
    rxLen := fbPort.RxLen;
    rx := fbPort.RxData;
    LastRxLen := rxLen;
    LastRx := rx;

    IF rxLen <> 9 THEN
        RxDiscardCount := RxDiscardCount + 1;
        LastDiscardId := 16#00030001; // passive discard: unexpected frame length
        CommOk := FALSE;
        CommErrorCount := CommErrorCount + 1;
        LastErrorId := LastDiscardId;
        RETURN;
    END_IF

    IF rx[0] <> SlaveId THEN
        RxDiscardCount := RxDiscardCount + 1;
        LastDiscardId := 16#00030002; // passive discard: wrong slave id
        CommOk := FALSE;
        CommErrorCount := CommErrorCount + 1;
        LastErrorId := LastDiscardId;
        RETURN;
    END_IF

    IF (rx[1] <> 3) OR (rx[2] <> 4) THEN
        RxDiscardCount := RxDiscardCount + 1;
        LastDiscardId := 16#00030003; // passive discard: unexpected function/byte count
        CommOk := FALSE;
        CommErrorCount := CommErrorCount + 1;
        LastErrorId := LastDiscardId;
        RETURN;
    END_IF

    crcRx := USINT_TO_WORD(rx[7]) OR SHL(USINT_TO_WORD(rx[8]), 8);
    crcCalc := F_ModbusCrc16(rx, 7);
    IF crcRx <> crcCalc THEN
        RxDiscardCount := RxDiscardCount + 1;
        LastDiscardId := 16#00030004; // passive discard: crc mismatch
        CommOk := FALSE;
        CommErrorCount := CommErrorCount + 1;
        LastErrorId := LastDiscardId;
        RETURN;
    END_IF

    high := SHL(USINT_TO_UINT(rx[3]), 8) OR USINT_TO_UINT(rx[4]);
    low := SHL(USINT_TO_UINT(rx[5]), 8) OR USINT_TO_UINT(rx[6]);
    IF WordSwap32 THEN
        high := SHL(USINT_TO_UINT(rx[5]), 8) OR USINT_TO_UINT(rx[6]);
        low := SHL(USINT_TO_UINT(rx[3]), 8) OR USINT_TO_UINT(rx[4]);
    END_IF

    uTmp := SHL(UINT_TO_UDINT(high), 16) OR UINT_TO_UDINT(low);
    dw := UDINT_TO_DWORD(uTmp);
    RelRaw := DWORD_TO_DINT(dw);
    RelMm := DINT_TO_LREAL(RelRaw) / 1000.0;
    AbsRaw := RelRaw;
    AbsMm := RelMm;

    CommOk := TRUE;
    LastErrorId := 0;
    LastDiscardId := 0;
END_IF

END_FUNCTION_BLOCK

// ---- POUs/FB_VibrationSensor.TcPOU
FUNCTION_BLOCK FB_VibrationSensor
VAR_INPUT
    Enable : BOOL;
    Channel : USINT;
    SlaveId : USINT;
    MinGapMs : UINT;
    TimeoutMs : UINT;
END_VAR
VAR_OUTPUT
    Busy : BOOL;
    PortReady : BOOL;
    CommOk : BOOL;
    CommErrorCount : UDINT;
    LastErrorId : UDINT;
    ExceptionCode : USINT;
    RxDiscardCount : UDINT;
    LastDiscardId : UDINT;
    SampleSeq : UDINT;

    AccXRaw : INT;
    AccYRaw : INT;
    AccZRaw : INT;
    VelXRaw : INT;
    VelYRaw : INT;
    VelZRaw : INT;
    TempRaw : INT;
    DispXRaw : INT;
    DispYRaw : INT;
    DispZRaw : INT;
    FreqXRaw : INT;
    FreqYRaw : INT;
    FreqZRaw : INT;

    AccX : LREAL;
    AccY : LREAL;
    AccZ : LREAL;
    VelX : LREAL;
    VelY : LREAL;
    VelZ : LREAL;
    TempC : LREAL;
    DispX : LREAL;
    DispY : LREAL;
    DispZ : LREAL;
    FreqX : LREAL;
    FreqY : LREAL;
    FreqZ : LREAL;

    LastTxLen : USINT;
    LastTx : ARRAY [0..21] OF USINT;
    LastRxLen : USINT;
    LastRx : ARRAY [0..21] OF USINT;
END_VAR
VAR
    mb : FB_ModbusRtuMaster;
    mbReqHold : BOOL;
    mbFunc : USINT;
    mbAddr : UINT;
    mbQty : USINT;
    mbWbc : USINT;
    mbWData : ARRAY [0..21] OF USINT;
    op : USINT;
    pollStep : USINT;
    minGapTime : TIME;
    timeoutTime : TIME;
    tmpI : INT;
END_VAR

IF NOT Enable THEN
    mbReqHold := FALSE;
    mbFunc := 0;
    mbAddr := 0;
    mbQty := 0;
    mbWbc := 0;
    op := 0;
    pollStep := 0;

    Busy := FALSE;
    PortReady := FALSE;
    CommOk := FALSE;
    LastErrorId := 0;
    ExceptionCode := 0;
    LastTxLen := 0;
    LastRxLen := 0;
    RETURN;
END_IF

IF MinGapMs = 0 THEN
    minGapTime := T#200ms;
ELSE
    minGapTime := UINT_TO_TIME(MinGapMs);
END_IF

IF TimeoutMs = 0 THEN
    timeoutTime := T#500ms;
ELSE
    timeoutTime := UINT_TO_TIME(TimeoutMs);
END_IF

mb(Enable := Enable,
   Channel := Channel,
   SlaveId := SlaveId,
   Req := mbReqHold,
   Func := mbFunc,
   Addr := mbAddr,
   Quantity := mbQty,
   WriteByteCount := mbWbc,
   WriteData := mbWData,
   Timeout := timeoutTime,
   MinGap := minGapTime);

PortReady := mb.PortReady;
Busy := mb.Busy;
ExceptionCode := mb.ExceptionCode;
RxDiscardCount := mb.RxDiscardCount;
LastDiscardId := mb.LastDiscardId;

IF mb.Busy THEN
    mbReqHold := FALSE;
END_IF

IF mb.TxLen > 0 THEN
    LastTxLen := mb.TxLen;
    LastTx := mb.TxFrame;
END_IF

IF mb.RxLen > 0 THEN
    LastRxLen := mb.RxLen;
    LastRx := mb.RxFrame;
END_IF

IF mb.Error THEN
    CommOk := FALSE;
    CommErrorCount := CommErrorCount + 1;
    LastErrorId := mb.ErrorId;
    op := 0;
    pollStep := 0;
END_IF

IF mb.Done THEN
    CommOk := TRUE;
    LastErrorId := 0;

    CASE op OF
    1: // 0x34..0x36 acceleration raw
        AccXRaw := WORD_TO_INT(UINT_TO_WORD(mb.ReadRegs[0]));
        AccYRaw := WORD_TO_INT(UINT_TO_WORD(mb.ReadRegs[1]));
        AccZRaw := WORD_TO_INT(UINT_TO_WORD(mb.ReadRegs[2]));
        AccX := INT_TO_LREAL(AccXRaw) / 32768.0 * 16.0;
        AccY := INT_TO_LREAL(AccYRaw) / 32768.0 * 16.0;
        AccZ := INT_TO_LREAL(AccZRaw) / 32768.0 * 16.0;

    2: // 0x3A..0x3C velocity raw
        VelXRaw := WORD_TO_INT(UINT_TO_WORD(mb.ReadRegs[0]));
        VelYRaw := WORD_TO_INT(UINT_TO_WORD(mb.ReadRegs[1]));
        VelZRaw := WORD_TO_INT(UINT_TO_WORD(mb.ReadRegs[2]));
        VelX := INT_TO_LREAL(VelXRaw) / 100.0;
        VelY := INT_TO_LREAL(VelYRaw) / 100.0;
        VelZ := INT_TO_LREAL(VelZRaw) / 100.0;

    3: // 0x40..0x46 temp/displacement/frequency raw
        TempRaw := WORD_TO_INT(UINT_TO_WORD(mb.ReadRegs[0]));
        DispXRaw := WORD_TO_INT(UINT_TO_WORD(mb.ReadRegs[1]));
        DispYRaw := WORD_TO_INT(UINT_TO_WORD(mb.ReadRegs[2]));
        DispZRaw := WORD_TO_INT(UINT_TO_WORD(mb.ReadRegs[3]));
        FreqXRaw := WORD_TO_INT(UINT_TO_WORD(mb.ReadRegs[4]));
        FreqYRaw := WORD_TO_INT(UINT_TO_WORD(mb.ReadRegs[5]));
        FreqZRaw := WORD_TO_INT(UINT_TO_WORD(mb.ReadRegs[6]));
        TempC := INT_TO_LREAL(TempRaw) / 100.0;
        DispX := INT_TO_LREAL(DispXRaw);
        DispY := INT_TO_LREAL(DispYRaw);
        DispZ := INT_TO_LREAL(DispZRaw);
        FreqX := INT_TO_LREAL(FreqXRaw) / 10.0;
        FreqY := INT_TO_LREAL(FreqYRaw) / 10.0;
        FreqZ := INT_TO_LREAL(FreqZRaw) / 10.0;
        SampleSeq := SampleSeq + 1;

    ELSE
        ;
    END_CASE

    op := 0;
    IF pollStep >= 3 THEN
        pollStep := 1;
    ELSE
        pollStep := pollStep + 1;
    END_IF
END_IF

IF (NOT mb.Busy) AND (op = 0) AND mb.PortReady AND (NOT mbReqHold) THEN
    IF pollStep = 0 THEN
        op := 1;
    ELSIF pollStep = 1 THEN
        op := 2;
    ELSIF pollStep = 2 THEN
        op := 3;
    ELSE
        op := 1;
    END_IF

    IF op = 1 THEN
        mbAddr := 16#0034;
        mbQty := 3;
    ELSIF op = 2 THEN
        mbAddr := 16#003A;
        mbQty := 3;
    ELSE
        mbAddr := 16#0040;
        mbQty := 7;
    END_IF

    mbFunc := 3;
    mbWbc := 0;
    mbReqHold := TRUE;
END_IF

END_FUNCTION_BLOCK
